FUNCTION "FC_WW_TELLER" : VOID
TITLE =
//$Revision: 1.56 $
//$Date: 2008/09/09 10:15:54CEST $
//$Author: schmoelp $
//
// Werkzeugwechsler Teller
AUTHOR : PS
FAMILY : DMC_H
NAME : WWPICKUP
VERSION : 0.0


VAR_INPUT
  gespannt : BOOL ;	// gespannt mit oder ohne Werkzeug
  gespannt_mWz : BOOL ;	// gespannt mit Werkzeug
  gespannt_oWz : BOOL ;	// gespannt ohne Werkzeug
  gespannt_Frg_Sp : BOOL ;	// gespannt mit Werkzeug Freigabe Spindeldrehen
  IB_MagKontr_aus : BOOL ;	//IB-Bit: Belegungskontrolle Magazin ausblenden
  AB_mit_Entriegeln : BOOL ;	//Ausbaustufe gesteuertes entriegeln im Magazin
  Frg_Service : BOOL ;	//Freigabe der Einzelbewegungen ohne Bedingung
  Bild_MAGEinstellung : BOOL ;
END_VAR
VAR_TEMP
  Klappe_auf_1 : BOOL ;
  Klappe_auf_2 : BOOL ;
  Vorbedingung_AF1 : BOOL ;
  Vorbedingung_AF2 : BOOL ;
  Vorbedingung_AF3 : BOOL ;
  PruefeAblageplatz : BOOL ;
  PruefeAbholplatz : BOOL ;
  ZvonPLC : BOOL ;
  IKZ_ausblasen : BOOL ;
  FC18_Error : BOOL ;
  Klappe_auf_BBK : BOOL ;
  Reset_Prgende : BOOL ;
  WV_laden_M1_aktiv : BOOL ;
  Schritt_gesetzt : BOOL ;
  Bild_WW_Handbedienung : BOOL ;
  MSST_Reset : BOOL ;
  WW_von_WZV : BOOL ;
  WZM_Fahrbefehl : BOOL ;
  BA_3_4 : BOOL ;
  F_ZHub_n_ausgefahren : BOOL ;
  F_ZHub_n_eingefahren : BOOL ;
  F_Mag_n_in_Position : BOOL ;
  F_Zange_n_auf : BOOL ;
  F_Zange_n_zu : BOOL ;
  F_Spanner_n_zu : BOOL ;
  F_Spanner_n_auf : BOOL ;
  F_Sp_n_gerichtet : BOOL ;
  F_MagKlappe_n_auf : BOOL ;
  F_MagKlappe_n_zu : BOOL ;
  F_Spindel_leer : BOOL ;
  F_VSP_Y_WW : BOOL ;
  HalterSp_auf : BOOL ;
  HalterSp_zu : BOOL ;
  PI_WZ_LS_GST : BOOL ;	//Positive Flanke Grundstellung Werkzeug entriegeln Ladestation
  FRG_WZ_MAN_RELEASE : BOOL ;
  Frg_Ventil_Hub : BOOL ;
  t_PI_T_quitt_Entladen : BOOL ;
  AB_WZB : BOOL ;	//mechanische Bruchkontrolle
  SFC12_RET_VAL : INT ;
  SFC12_SRCBLK : INT ;
  SFC12_DSTBLK : INT ;
  Achssperre : BOOL ;
  NewToolTx : BOOL ;
  NewToolT0 : BOOL ;
  OldToolTx : BOOL ;
  OldToolT0 : BOOL ;
  Schritt_vorwaerts : BOOL ;	//Schrittkette vorwärts
  Schritt_rueckwaerts : BOOL ;	//Schrittkette rückwärts
  Taste_vorwaerts : BOOL ;
  Taste_rueckwaerts : BOOL ;
  PI_T_vorwaerts : BOOL ;
  PI_T_rueckwaerts : BOOL ;
  EB_Frg_Klappe_auf : BOOL ;
  EB_Klappe_auf : BOOL ;
  EB_Frg_Klappe_zu : BOOL ;
  EB_Klappe_zu : BOOL ;
  EB_Frg_Wz_aus : BOOL ;
  EB_Frg_Wz_ein : BOOL ;
  EB_Frg_entspannen : BOOL ;
  EB_entspannen : BOOL ;
  EB_Frg_spannen : BOOL ;
  EB_spannen : BOOL ;
  EB_Frg_KR_einfahren : BOOL ;
  EB_KR_einfahren : BOOL ;
  EB_Frg_KR_ausfahren : BOOL ;
  EB_KR_ausfahren : BOOL ;
  EB_Frg_X_WWPos : BOOL ;
  EB_Frg_X_WartePos : BOOL ;
  EB_Hand_WW : BOOL ;
  Handbetrieb : BOOL ;
  Achse_angewaehlt : BOOL ;
  PI_Start_KR : BOOL ;
  Temp_INT : INT ;
  VSP_M_Wechsler : BOOL ;
  VSP_M_KR_GRSTn : BOOL ;
  VSP_M_Ls_GRSTn : BOOL ;
  VSP_M_BBK : BOOL ;
  VSP_M_aus_n : BOOL ;
  EB_Taste_steht_an : BOOL ;
  FC21_Error : BOOL ;
  t_AxFrg_y : BOOL ;
  t_Fahrbefehl_y : BOOL ;
  TX_O_WW_1_ZYL_GST : BOOL ;
  TX_O_WW_1_ZYL_SPI : BOOL ;
  A_DPR : ARRAY  [0 .. 15 ] OF BOOL ;
  FC21_ErrCode : INT ;
END_VAR
BEGIN
NETWORK
TITLE ============ allgemeine Signale ==============
// Netzwerk-Übersicht
// ==================
// NW 1: =========== allgemeine Signale ==============
// NW 2: Ausbaustufe mechanische Werkzeugbruchkontrolle
// NW 3: Taste Reset oder Programmende
// NW 4: Betriebsart 3, 4
// NW 5: JOG-Betrieb
// NW 6: Bildanwahl Einzelbewegung
// NW 7: Bildanwahl Semifunktion
// NW 8: Zange geöffnet
// NW 9: Zange geschlossen
// NW 10: Fahrbefehl Werkzeugmagazin steht an
// NW 11: ========== Signale von Werkzeugverwalung ==============
// NW 12: WZV: Werkzeugwechsel steht an
// NW 13: WZV: Aufgerufenes Werkzeug Tx
// NW 14: WZV: Aufgerufenes Werkzeug T0
// NW 15: WZV: Spindel belegt
// NW 16: WZV: Spindel leer
// NW 17: WZV: Vorbedingung Folge 1 Tx M6 Spindel leer
// NW 18: WZV: Vorbedingung Folge 2 Tx M6 Spindel belegt
// NW 19: WZV: Vorbedingung Folge 3 T0 M6 Spindel belegt
// NW 20: ============= Kegelreinigung ==================
// NW 21: KR: Einzelbewegung Freigabe einfahren
// NW 22: KR: Einzelbewegung einfahren
// NW 23: KR: Einzelbewegung Freigabe ausfahren
// NW 24: KR: Einzelbewegung ausfahren
// NW 25: KR: Einzelbewegung ausfahren speichern
// NW 26: KR: Einzelbewegung Ansteuerung Anzeige
// NW 27: Überwachung Kegelreinigung
// NW 28: KR: Start Werkzeug reinigen Tellermagazin
// NW 29: KR: aus-/einfahren
// NW 30: KR: Ausgang ausfahren
// NW 31: KR: Zeit starten
// NW 32: KR: beendet
// NW 33: ============== Werkzeugwechsel ===============
// NW 34: WW: Zyklus L6 wurde gestartet
// NW 35: WW: rücksetzen
// NW 36: WW: Auswertung Schritt gesetzt
// NW 37: WW: START
// NW 38: WW: Rücksetzen M-Funktion M06
// NW 39: WZW: Aktiver Ablauf
// NW 40: WW: 2nd software limit switch plus
// NW 41: WW: Folge 1 Tx M6 Spindel leer / Auftrag 1
// NW 42: WW: Folge 1 Freigabe fahre ins Magazin
// NW 43: WW: Folge 1 Auftrag 2: Einwechseln neues Werkzeug
// NW 44: WW: Folge 1 Tx M6 Spindel leer beendet
// NW 45: WW: Folge 2 Tx M6 Spindel belegt / Auftrag 3
// NW 46: WW: Folge 2 Freigabe fahre ins Magazin
// NW 47: WW: Folge 2 HILFSSCHRITT2
// NW 48: WW: Folge 2 Auftrag 2: Einwechseln neues Werkzeug
// NW 49: WW: Folge 2 beendet
// NW 50: WW: Folge 3 T0 M6 Spindel belegt / Auftrag 3
// NW 51: WW: Folge 3 Freigabe fahre ins Magazin
// NW 52: WW: Folge 3 Einwechseln kein Werkzeug
// NW 53: WW: Folge 3 beendet
// NW 54: WW: ABBRUCH -> FREIFAHREN
// NW 55: Taste Werkzeugwechsler vorwärts in Grundstellung fahren
// NW 56: Taste Werkzeugwechsler rückwärts in Grundstellung fahren
// NW 57: WW: Vorwärts Taste
// NW 58: WW: Rückwärts Taste
// NW 59: WW: Freigabe VOR/ZURUECK Freifahren
// NW 60: WW: Vorwärts Flanke Taste
// NW 61: WW: Vorwärts Bewegung
// NW 62: WW: Vorwärts Schrittkette
// NW 63: WW: Rückwärts Flanke Taste
// NW 64: WW: Rückwärts Bewegung
// NW 65: WW: Rückwärts gespeichert
// NW 66: WW: Rückwärts Schrittkette
// NW 67: WW: FREIGABE AUSGAENGE FUER ABLAUF
// NW 68: WW: ANZEIGE VORWAERTS
// NW 69: WW: ANZEIGE RUECKWAERTS
// NW 70: WW: Semifunktion Ansteuerung Anzeige Werkzeugwechsler
// NW 71: WW: initialisieren
// NW 72: WW: SCHRITT_0 GRUNDSTELLUNG
// NW 73: WW: GRUNDSTELLUNG MELDEN
// NW 74: WW: Grundstellung Werkzeugwechsler
// NW 75: WW: Werkzeugwechsel beendet an andere Module
// NW 76: WW: SCHRITT_1
// NW 77: WW: SCHRITT_2
// NW 78: WW: SCHRITT_3
// NW 79: WW: SCHRITT_4
// NW 80: WW: Datentausch ablegen
// NW 81: WW: SCHRITT_5
// NW 82: WW: SCHRITT_6
// NW 83: WW: SCHRITT_7 SONDERSCHRITT
// NW 84: WW: Rücksetzen Auftrag 1 und 3
// NW 85: WW: SCHRITT_8
// NW 86: WW: SCHRITT_9
// NW 87: WW: Datentausch aufnehmen
// NW 88: WW: SCHRITT_10
// NW 89: WW: SCHRITT_11
// NW 90: WW: Rücksetzen Schritt 10
// NW 91: WW: SCHRITT_12
// NW 92: WW: Prüfen, ob Ablageplatz im Magazin leer ist
// NW 93: WW: Prüfen, ob Abholplatz im Magazin belegt ist
// NW 94: WW: Magazinplatz Belegung kontrolliert und i.O.
// NW 95: =========== Magazinklappe (Werkzeugwechslertür) =============
// NW 96: WWT: öffnen mit Freigabe
// NW 97: WWT: öffnen ohne Freigabe
// NW 98: WWT: Einzelbewegung Freigabe öffnen
// NW 99: WWT: Einzelbewegung öffnen
// NW 100: WWT: Einzelbewegung Freigabe schliessen
// NW 101: WWT: Einzelbewegung schliessen
// NW 102: WWT: Einzelbewegung öffnen speichern
// NW 103: WWT: Einzelbewegung schliessen speichern
// NW 104: WWT: Einzelbewegung Ansteuerung Anzeige
// NW 105: HMI-Bild 35 (WZW7): WWT: Einzelbewegung Ansteuerung Anzeige
// NW 106: WWT: Ausgang öffnen
// NW 107: WWT: Ausgang schliessen
// NW 108: WWT: Ausgang schliessen Reset M272
// NW 109: WWT: Reset Ausgang schliessen
// NW 110: ========== Werkzeug in / aus Spindel ===============
// NW 111: WZHUB: BEFEHL FAHRE auf AUSFAHRPOSITION
// NW 112: WZHUB: BEFEHL FAHRE WW-Achse auf Einfahrposition
// NW 113: Hub in Spindelstellung
// NW 114: Hub in Grundstellung
// NW 115: WZHUB: Einzelbewegung Freigabe Werkzeug Spindel aus- einfahren
// NW 116: WZHUB: Einzelbewegung Werkzeug aus Spindel ausfahren
// NW 117: WZHUB: Einzelbewegung WW-Achse auf Einfahrposition
// NW 118: WZHUB: Reset Einzelbewegung WW-Achse wenn nicht in Position
// NW 119: WZHUB: Freigabe Ansteuerung Ventil Hub ein- / ausfahren
// NW 120: WZHUB: Ventil Hub einfahren
// NW 121: WZHUB: Ventil Hub ausfahren
// NW 122: WZHUB: (WZW1) Einzelbewegung Ansteuerung Anzeige
// NW 123: WZHUB: (WZW7) Einzelbewegung Ansteuerung Anzeige
// NW 124: =========== Spindel in / aus Werkzeugwechsler ============
// NW 125: X-Achse: Befehl auf Warteposition fahren
// NW 126: X-Achse: Befehl auf Wechselposition fahren
// NW 127: X-Achse: Einzelbewegung Freigabe auf Warteposition
// NW 128: X-Achse: Einzelbewegung auf Warteposition fahren
// NW 129: X-Achse: Einzelbewegung Freigabe auf Wechselposition
// NW 130: X-Achse: Einzelbewegung auf Wechselposition fahren
// NW 131: X-Achse: Einzelbewegung Ansteuerung Anzeige
// NW 132: Y-Achse: Freigabe
// NW 133: Y-Achse: Fahrbefehl
// NW 134: Y-Achse: HMI Rettung
// NW 135: Spindel: Befehl auf Werkzeugwechselposition
// NW 136: Spindel: HMI Rettung
// NW 137: ======== Werkzeug im Magazin entsichern Wechselstelle ========
// NW 138: WW_MagTasche: BEFEHL Werkzeug entsichern Spindelseite
// NW 139: WW_MagTasche: Ausgang Werkzeug entsichern Spindelseite
// NW 140: ======== Werkzeug im Magazin entsichern Ladestelle ========
// NW 141: WM_MagTasche: Ausgang Werkzeug entsichern an BELADESTATION
// NW 142: WM_MagTasche: Werkzeug wurde an BELADESTATION entsichert
// NW 143: ========= Werkzeug entspannen im Ablauf ===========
// NW 144: WZ-Spanner: Einzelbewegung Freigabe Werkzeug entspannen
// NW 145: WZ-Spanner: Einzelbewegung Werkzeug entspannen
// NW 146: WZ-Spanner: Einzelbewegung Freigabe Werkzeug spannen
// NW 147: WZ-Spanner: Einzelbewegung Werkzeug spannen
// NW 148: WZ-Spanner: Einzelbewegung Ansteuerung Anzeige
// NW 149: WZ-Spanner: Einzelbewegung Ansteuerung Anzeige
// NW 150: WZ-Spanner: BEFEHL WZ ENTSPANNEN
// NW 151: WZ-Spanner: BEFEHL WZ SPANNEN
// NW 152: WZ-Spanner: Ausgang Spanner öffnen
// NW 153: Ausgang SPINDELKONUS AUSBLASEN
// NW 154: Positive Flanke Taste quittieren Entladen
// NW 155: Pneumatikzyl. Verriegelung WZ lösen
// NW 156: Pneumatikzyl. Verriegelung WZ verriegeln
// NW 157: ========= Vorschubsperren ===============
// NW 158: VSP, alle Achsen
// NW 159: VSP-X, Werkzeugwechsler
// NW 160: _701303 Vorschubsperre X Werkzeugwechsler
// NW 161: VSP-Y, Werkzeugwechsler
// NW 162: Fehler Vorschubsperre Y Werkzeugwechsler
// NW 163: VSP-Z, Werkzeugwechsler
// NW 164: _701305 Vorschubsperre Z Werkzeugwechsler
// NW 165: VSP-M, Bohrerbruchkontrolle nicht in Grundstellung
// NW 166: VSP-M, Magazin nicht in Position aus Spindel ausgefahren
// NW 167: VSP-M, Werkzeugwechsler
// NW 168: VSP-M, Waschstation nicht in Grundstellung
// NW 169: Positive Flanke Grundstellung Werkzeug entriegeln Ladestation
// NW 170: Werkzeug wurde richtig eingelegt
// NW 171: VSP-M, Werkzeug in Ladestation nicht gesichert
// NW 172: VSP-M, Werkzeugwechsler
// NW 173: VSP-M, Verzögerung Fehlermeldung
// NW 174: 701306 "MEL, Vorschubsperre Magazin Werkzeugwechsler"
// NW 175: 701307 Vorschubsperre Magazin Waschstation nicht in Grundst
// NW 176: 701308 VSP Magazin Bohrerbruchkontrolle nicht in Grundstellung
// NW 177: 701309 VSP, Magazin nicht in Position aus Spindel ausgefahren
// NW 178: 700363 Warnung: Werkzeug in Ladestation nicht gesichert
// NW 179: 511214: Meldung: Werkzeug in Ladestation nicht gesichert
// NW 180: _700434 VS-H, ENDSCHALTERSTOERUNG Werkzeugwechsel
// NW 181: ============ Überwachung Endposition ==========
// NW 182: Fehler MAGAZIN NICHT AUSGEFAHREN
// NW 183: Fehler MAGAZIN NICHT EINGEFAHREN
// NW 184: Fehler MAGAZIN NICHT IN POSITION
// NW 185: Fehler WZ-ZANGE NICHT OFFEN
// NW 186: Fehler WZ-ZANGE NICHT GESCHLOSSEN
// NW 187: Fehler WZ-SPANNER NICHT GESPANNT
// NW 188: Fehler WZ-SPANNER NICHT GELOEST
// NW 189: Fehler SPINDEL NICHT GERICHTET
// NW 190: Fehler Magazinklappe nicht geöffnet
// NW 191: Fehler Magazinklappe nicht geschlossen
// NW 192: Fehler Spindel leer
// NW 193: gespeicherte Fehlermeldungen löschen
// NW 194: WZW nicht erlaubt
// NW 195: Start Wartezeit für Endlagenkontrolle
// NW 196: Wartezeit für Endlagenkontrolle abgelaufen ?
// NW 197: _700355 Werkzeugmagazin nicht ausgefahren
// NW 198: _700356 Werkzeugmagazin nicht eingefahren
// NW 199: _700361 Magazin nicht in Position
// NW 200: _700354 Werkzeug im Magazin nicht entsichert
// NW 201: _700362 Werkzeug in Magazin nicht gesichert
// NW 202: _700353 Werkzeug in Spindel nicht gespannt
// NW 203: _700351 Werkzeug in Spindel nicht entspannt
// NW 204: _700360 Spindel nicht gerichtet
// NW 205: _700357 Magazinklappe nicht geöffnet
// NW 206: _700358 Magazinklappe nicht geschlossen
// NW 207: _701302 Spindel leer
// NW 208: _701304 VSP-Y Werkzeugwechsler
// NW 209: ======== Sonstige Fehler- Betriebsmeldungen ===========
// NW 210: _700348 Magazinplatz/Greifer belegt
// NW 211: _700349 Magazinplatz/Greifer leer
// NW 212: _700350 Ladestation nicht geschlossen
// NW 213: _701321 Spindel belegt
// NW 214: _700352 Werkzeug Be- oder Entladen aktiv
// NW 215: Taste für Einzelbewegung Achsen betätigt
// NW 216: _700550 EINLESESPERRE, Werkzeugwechsel
// NW 217: ======== ASUP Einzelbewegung Achsen ========
// NW 218: ASUP-EB: Schnittstelle Dual-Port-RAM 16.0
// NW 219: ASUP-EB: Schnittstelle Dual-Port-RAM 16.1
// NW 220: ASUP-EB: Schnittstelle Dual-Port-RAM 16.2
// NW 221: ASUP-EB: Schnittstelle Dual-Port-RAM 16.3
// NW 222: ASUP-EB: Schnittstelle Dual-Port-RAM 16.4
// NW 223: Asup abbrechen wenn Taste wieder losgelassen wird
// NW 224: Eingang "MSSTstReset" auf "1" zuweisen
// NW 225: ASUP-Rettung: Werkzeugwechsler automatisch in Grundstellung
// NW 226: ASUP-EB: Schnittstelle Dual-Port-RAM nicht benutzte Bits
// NW 227: ASUP-EB: Aufruf Kanal-DB für FC21
// NW 228: ASUP-EB: Übergabe an DUAL-PORT-RAM
// NW 229: ASUP-EB: Start für Einzelbewegung Achsen
// NW 230: GRundstelltung Radmagazin
// NW 231: ============ Signale an andere Module =============
// NW 232: Übergabe der Schrittnummer Werkzeugwechsel an HMI
// NW 233: An NC: PLC-Freigabe Werkzeugwechsel
// NW 234: An NC: Rad in Wechselstellung nach Be./Enladen an Beladestelle
//
      NOP   0;

NETWORK
TITLE =Ausbaustufe mechanische Werkzeugbruchkontrolle
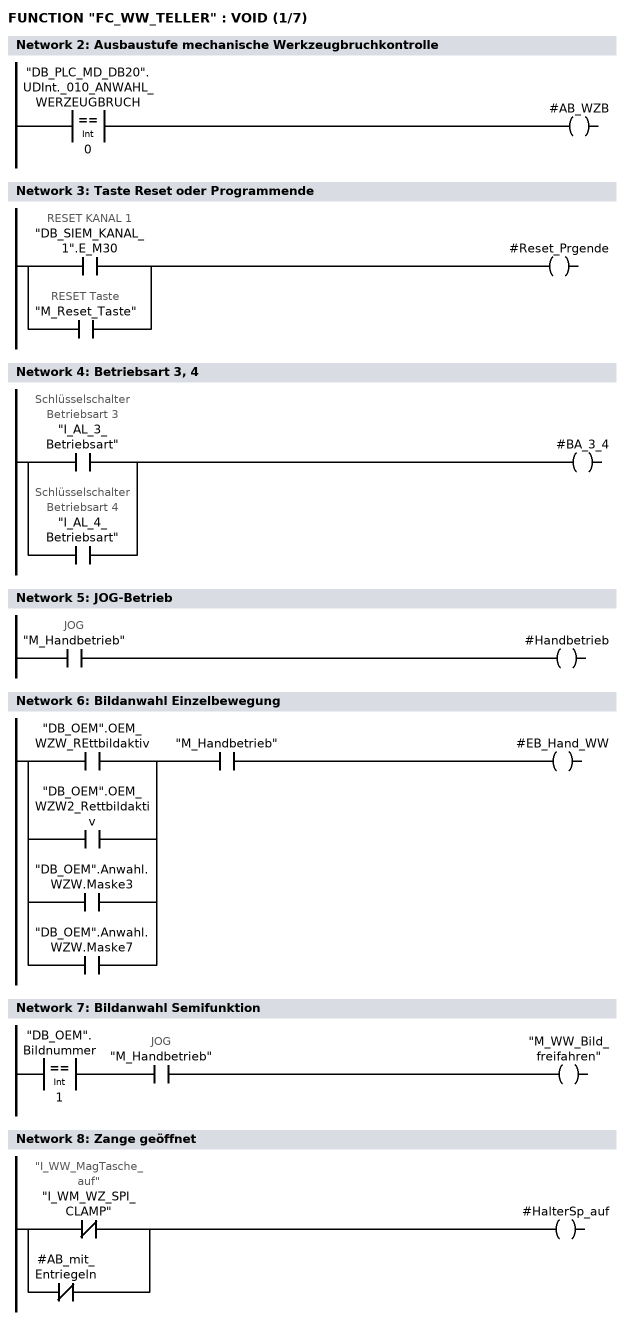

      L     "DB_PLC_MD_DB20".UDInt._010_ANWAHL_WERZEUGBRUCH;
      L     0;
      ==I   ;
      =     #AB_WZB;
NETWORK
TITLE =Taste Reset oder Programmende

      O     "DB_SIEM_KANAL_1".E_M30; // RESET KANAL 1
      O     "M_Reset_Taste"; // RESET Taste
      =     #Reset_Prgende;

NETWORK
TITLE =Betriebsart 3, 4

      O     "I_AL_3_Betriebsart"; // Schlüsselschalter Betriebsart 3
      O     "I_AL_4_Betriebsart"; // Schlüsselschalter Betriebsart 4
      =     #BA_3_4;


NETWORK
TITLE =JOG-Betrieb

      U     "M_Handbetrieb"; // JOG
      =     #Handbetrieb;

NETWORK
TITLE =Bildanwahl Einzelbewegung
//
      U(    ;
      O     "DB_OEM".OEM_WZW_REttbildaktiv;
      O     "DB_OEM".OEM_WZW2_Rettbildaktiv;
      O     "DB_OEM".Anwahl.WZW.Maske3;
      O     "DB_OEM".Anwahl.WZW.Maske7;
      )     ; // JOG
      U     "M_Handbetrieb";

      =     #EB_Hand_WW;
NETWORK
TITLE =Bildanwahl Semifunktion

      U(    ;
      L     "DB_OEM".Bildnummer;
      L     1;
      ==I   ;
      )     ;
      U     "M_Handbetrieb"; // JOG
      =     "M_WW_Bild_freifahren";

NETWORK
TITLE =Zange geöffnet

      ON    "I_WM_WZ_SPI_CLAMP"; //"I_WW_MagTasche_auf"
      ON    #AB_mit_Entriegeln;
      =     #HalterSp_auf;

NETWORK
TITLE =Zange geschlossen
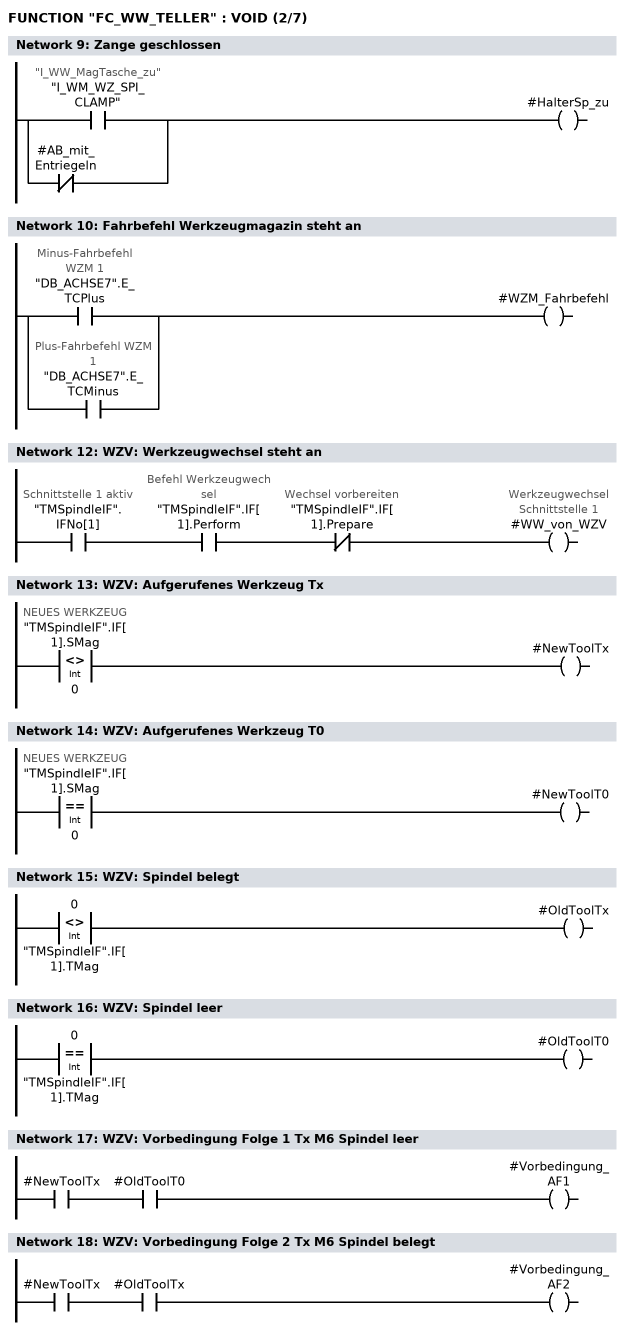

      O     "I_WM_WZ_SPI_CLAMP"; //"I_WW_MagTasche_zu"
      ON    #AB_mit_Entriegeln;
      =     #HalterSp_zu;

NETWORK
TITLE =Fahrbefehl Werkzeugmagazin steht an

      O     "DB_ACHSE7".E_TCPlus; // Minus-Fahrbefehl WZM 1
      O     "DB_ACHSE7".E_TCMinus; // Plus-Fahrbefehl WZM 1
      =     #WZM_Fahrbefehl;

NETWORK
TITLE =========== Signale von Werkzeugverwalung ==============



NETWORK
TITLE =WZV: Werkzeugwechsel steht an

      U     "TMSpindleIF".IFNo[1]; // Schnittstelle 1 aktiv
      U     "TMSpindleIF".IF[1].Perform; // Befehl Werkzeugwechsel
      UN    "TMSpindleIF".IF[1].Prepare; // Wechsel vorbereiten
      =     #WW_von_WZV; // Werkzeugwechsel Schnittstelle 1

NETWORK
TITLE =WZV: Aufgerufenes Werkzeug Tx

      L     "TMSpindleIF".IF[1].SMag; // NEUES WERKZEUG
      L     0;
      <>I   ;
      =     #NewToolTx;

NETWORK
TITLE =WZV: Aufgerufenes Werkzeug T0

      L     "TMSpindleIF".IF[1].SMag; // NEUES WERKZEUG
      L     0;
      ==I   ;
      =     #NewToolT0;

NETWORK
TITLE =WZV: Spindel belegt

      L     0;
      L     "TMSpindleIF".IF[1].TMag; // ALTES WERKZEUG
      <>I   ;
      =     #OldToolTx;

NETWORK
TITLE =WZV: Spindel leer

      L     0;
      L     "TMSpindleIF".IF[1].TMag; // ALTES WERKZEUG
      ==I   ;
      =     #OldToolT0;

NETWORK
TITLE =WZV: Vorbedingung Folge 1 Tx M6 Spindel leer

      U     #NewToolTx;
      U     #OldToolT0;
      =     #Vorbedingung_AF1;

NETWORK
TITLE =WZV: Vorbedingung Folge 2 Tx M6 Spindel belegt

      U     #NewToolTx;
      U     #OldToolTx;
      =     #Vorbedingung_AF2;
NETWORK
TITLE =WZV: Vorbedingung Folge 3 T0 M6 Spindel belegt
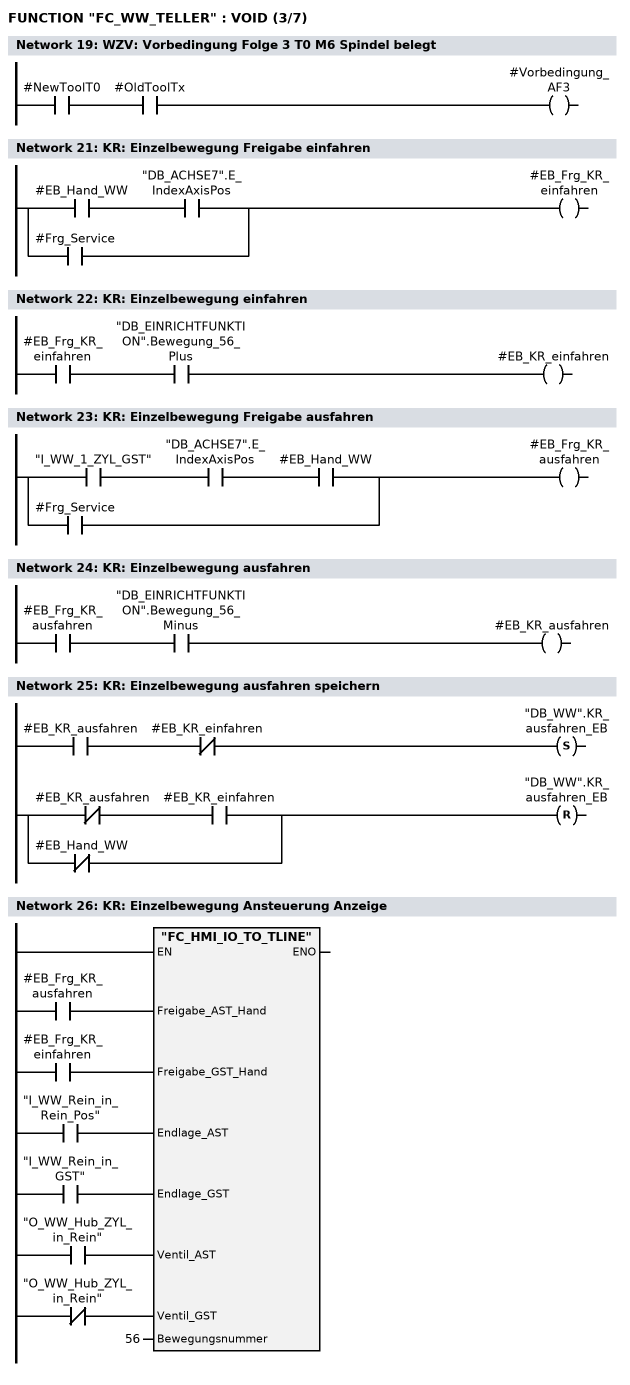

      U     #NewToolT0;
      U     #OldToolTx;
      =     #Vorbedingung_AF3;
NETWORK
TITLE ============== Kegelreinigung ==================



NETWORK
TITLE =KR: Einzelbewegung Freigabe einfahren

      U     #EB_Hand_WW;
      U     "DB_ACHSE7".E_IndexAxisPos;
      O     #Frg_Service;
      =     #EB_Frg_KR_einfahren;

NETWORK
TITLE =KR: Einzelbewegung einfahren

      U     #EB_Frg_KR_einfahren;
      U     "DB_EINRICHTFUNKTION".Bewegung_56_Plus;
      =     #EB_KR_einfahren;

NETWORK
TITLE =KR: Einzelbewegung Freigabe ausfahren

      U     "I_WW_1_ZYL_GST";
      U     "DB_ACHSE7".E_IndexAxisPos;
      U     #EB_Hand_WW;
      O     #Frg_Service;
      =     #EB_Frg_KR_ausfahren;
NETWORK
TITLE =KR: Einzelbewegung ausfahren

      U     #EB_Frg_KR_ausfahren;
      U     "DB_EINRICHTFUNKTION".Bewegung_56_Minus;
      =     #EB_KR_ausfahren;

NETWORK
TITLE =KR: Einzelbewegung ausfahren speichern

      U     #EB_KR_ausfahren;
      UN    #EB_KR_einfahren;
      S     "DB_WW".KR_ausfahren_EB;

      U(    ;
      UN    #EB_KR_ausfahren;
      U     #EB_KR_einfahren;
      ON    #EB_Hand_WW;
      )     ;
      R     "DB_WW".KR_ausfahren_EB;
      NOP   0;

NETWORK
TITLE =KR: Einzelbewegung Ansteuerung Anzeige

      U     #EB_Frg_KR_ausfahren;
      =     L     24.0;
      BLD   103;
      U     #EB_Frg_KR_einfahren;
      =     L     24.1;
      BLD   103;
      U     "I_WW_Rein_in_Rein_Pos";
      =     L     24.2;
      BLD   103;
      U     "I_WW_Rein_in_GST";
      =     L     24.3;
      BLD   103;
      U     "O_WW_Hub_ZYL_in_Rein";
      =     L     24.4;
      BLD   103;
      UN    "O_WW_Hub_ZYL_in_Rein";
      =     L     24.5;
      BLD   103;
      CALL "FC_HMI_IO_TO_TLINE" (
           Freigabe_AST_Hand        := L     24.0,
           Freigabe_GST_Hand        := L     24.1,
           Endlage_AST              := L     24.2,
           Endlage_GST              := L     24.3,
           Ventil_AST               := L     24.4,
           Ventil_GST               := L     24.5,
           Bewegungsnummer          := 56);
      NOP   0;
NETWORK
TITLE =Überwachung Kegelreinigung
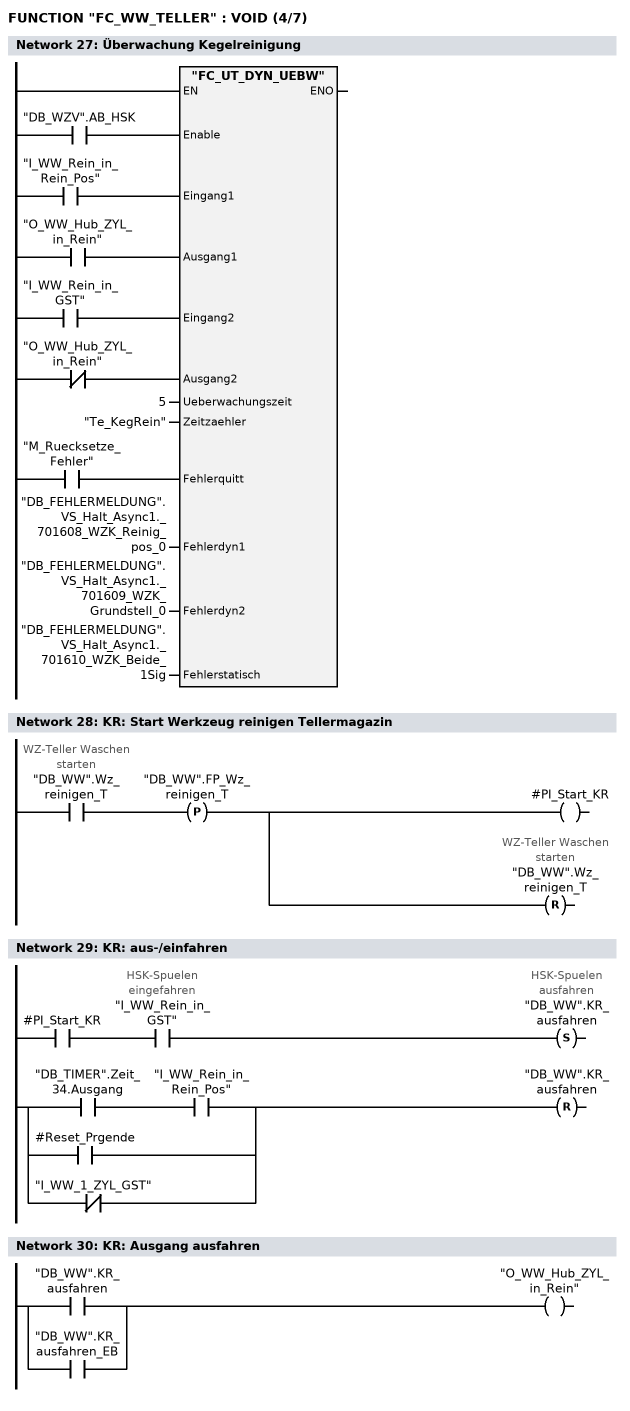

      U     "DB_WZV".AB_HSK;
      =     L     24.0;
      BLD   103;
      U     "I_WW_Rein_in_Rein_Pos";
      =     L     24.1;
      BLD   103;
      U     "O_WW_Hub_ZYL_in_Rein";
      =     L     24.2;
      BLD   103;
      U     "I_WW_Rein_in_GST";
      =     L     24.3;
      BLD   103;
      UN    "O_WW_Hub_ZYL_in_Rein";
      =     L     24.4;
      BLD   103;
      U     "M_Ruecksetze_Fehler";
      =     L     24.5;
      BLD   103;
      CALL "FC_UT_DYN_UEBW" (
           Enable                   := L     24.0,
           Eingang1                 := L     24.1,
           Ausgang1                 := L     24.2,
           Eingang2                 := L     24.3,
           Ausgang2                 := L     24.4,
           Ueberwachungszeit        := 5,
           Zeitzaehler              := "Te_KegRein",
           Fehlerquitt              := L     24.5,
           Fehlerdyn1               := "DB_FEHLERMELDUNG".VS_Halt_Async1._701608_WZK_Reinig_pos_0,
           Fehlerdyn2               := "DB_FEHLERMELDUNG".VS_Halt_Async1._701609_WZK_Grundstell_0,
           Fehlerstatisch           := "DB_FEHLERMELDUNG".VS_Halt_Async1._701610_WZK_Beide_1Sig);
      NOP   0;
NETWORK
TITLE =KR: Start Werkzeug reinigen Tellermagazin

      U     "DB_WW".Wz_reinigen_T; // WZ-Teller Waschen starten
      FP    "DB_WW".FP_Wz_reinigen_T; // PF: WZ waschen Start
      =     #PI_Start_KR;
      R     "DB_WW".Wz_reinigen_T; // WZ-Teller Waschen starten

NETWORK
TITLE =KR: aus-/einfahren

      U     #PI_Start_KR;
      U     "I_WW_Rein_in_GST"; // HSK-Spuelen eingefahren
      S     "DB_WW".KR_ausfahren; // HSK-Spuelen ausfahren

      U(    ;
      U     "DB_TIMER".Zeit_34.Ausgang;
      U     "I_WW_Rein_in_Rein_Pos";
      O     #Reset_Prgende;

      ON    "I_WW_1_ZYL_GST";
      )     ;
      R     "DB_WW".KR_ausfahren;
      NOP   0;
NETWORK
TITLE =KR: Ausgang ausfahren

      O     "DB_WW".KR_ausfahren;
      O     "DB_WW".KR_ausfahren_EB;
      =     "O_WW_Hub_ZYL_in_Rein";

NETWORK
TITLE =KR: Zeit starten
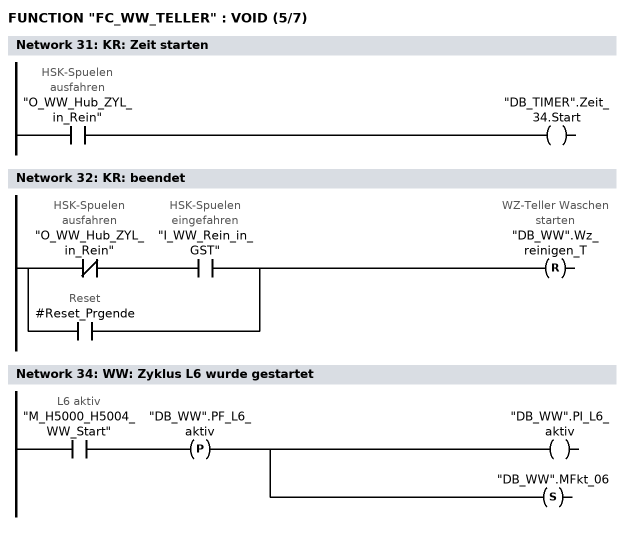

      U     "O_WW_Hub_ZYL_in_Rein"; // HSK-Spuelen ausfahren
      =     "DB_TIMER".Zeit_34.Start;

NETWORK
TITLE =KR: beendet

      UN    "O_WW_Hub_ZYL_in_Rein"; // HSK-Spuelen ausfahren
      U     "I_WW_Rein_in_GST"; // HSK-Spuelen eingefahren
      O     #Reset_Prgende; //Reset
      R     "DB_WW".Wz_reinigen_T; // WZ-Teller Waschen starten

NETWORK
TITLE =============== Werkzeugwechsel ===============



NETWORK
TITLE =WW: Zyklus L6 wurde gestartet

      U     "M_H5000_H5004_WW_Start"; // L6 aktiv
      FP    "DB_WW".PF_L6_aktiv;
      =     "DB_WW".PI_L6_aktiv;
      S     "DB_WW".MFkt_06;

NETWORK
TITLE =WW: rücksetzen
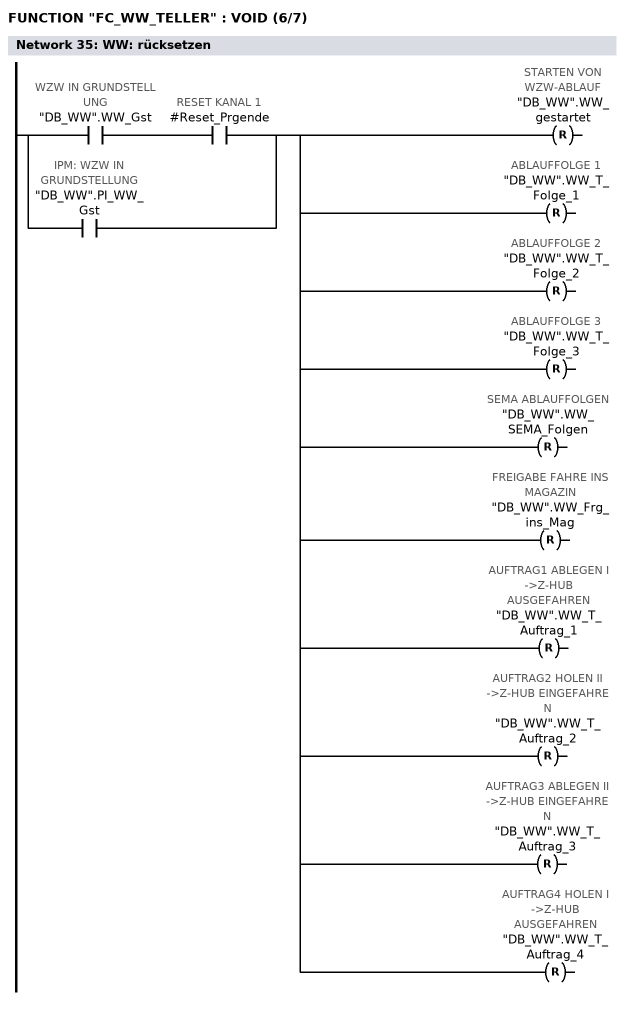

      U     "DB_WW".WW_Gst; // WZW IN GRUNDSTELLUNG
      U     #Reset_Prgende; // RESET KANAL 1
      O     "DB_WW".PI_WW_Gst; // IPM: WZW IN GRUNDSTELLUNG
      R     "DB_WW".WW_gestartet; // STARTEN VON WZW-ABLAUF
      R     "DB_WW".WW_T_Folge_1; // ABLAUFFOLGE 1
      R     "DB_WW".WW_T_Folge_2; // ABLAUFFOLGE 2
      R     "DB_WW".WW_T_Folge_3; // ABLAUFFOLGE 3
      R     "DB_WW".WW_SEMA_Folgen; // SEMA ABLAUFFOLGEN
      R     "DB_WW".WW_Frg_ins_Mag; // FREIGABE FAHRE INS MAGAZIN
      R     "DB_WW".WW_T_Auftrag_1; // AUFTRAG1 ABLEGEN I ->Z-HUB AUSGEFAHREN
      R     "DB_WW".WW_T_Auftrag_2; // AUFTRAG2 HOLEN II ->Z-HUB EINGEFAHREN
      R     "DB_WW".WW_T_Auftrag_3; // AUFTRAG3 ABLEGEN II ->Z-HUB EINGEFAHREN
      R     "DB_WW".WW_T_Auftrag_4; // AUFTRAG4 HOLEN I ->Z-HUB AUSGEFAHREN

NETWORK
TITLE =WW: Auswertung Schritt gesetzt
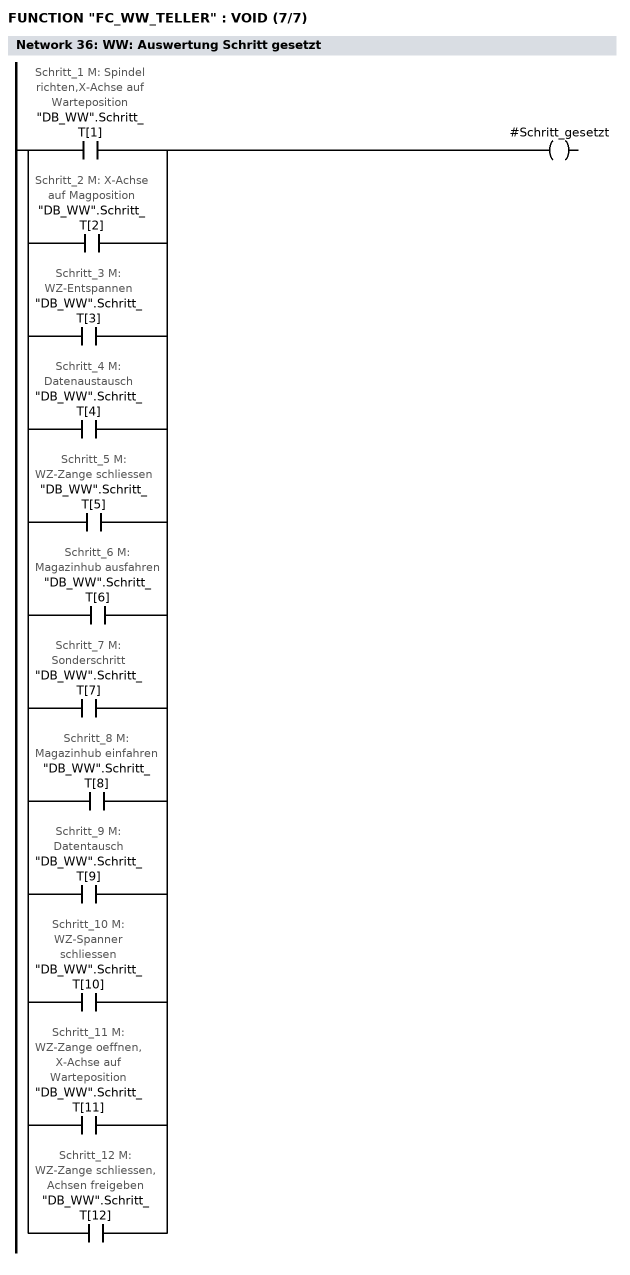

      O     "DB_WW".Schritt_T[1]; // Schritt_1 M: Spindel richten,X-Achse auf Warteposition
      O     "DB_WW".Schritt_T[2]; // Schritt_2 M: X-Achse auf Magposition
      O     "DB_WW".Schritt_T[3]; // Schritt_3 M: WZ-Entspannen
      O     "DB_WW".Schritt_T[4]; // Schritt_4 M: Datenaustausch
      O     "DB_WW".Schritt_T[5]; // Schritt_5 M: WZ-Zange schliessen
      O     "DB_WW".Schritt_T[6]; // Schritt_6 M: Magazinhub ausfahren
      O     "DB_WW".Schritt_T[7]; // Schritt_7 M: Sonderschritt
      O     "DB_WW".Schritt_T[8]; // Schritt_8 M: Magazinhub einfahren
      O     "DB_WW".Schritt_T[9]; // Schritt_9 M: Datentausch
      O     "DB_WW".Schritt_T[10]; // Schritt_10 M: WZ-Spanner schliessen
      O     "DB_WW".Schritt_T[11]; // Schritt_11 M: WZ-Zange oeffnen, X-Achse auf Warteposition
      O     "DB_WW".Schritt_T[12]; // Schritt_12 M: WZ-Zange schliessen, Achsen freigeben
      =     #Schritt_gesetzt;

NETWORK
TITLE =WW: START

      UN(   ;
      U(    ;
      L     "TMSpindleIF".IF[1].SMag; // NEUES WERKZEUG
      L     9999;
      ==I   ;
      )     ;
      U(    ;
      L     "TMSpindleIF".IF[1].TMag; // ALTES WERKZEUG
      L     0;
      ==I   ;
      )     ;
      O     ;
      U(    ;
      L     "TMSpindleIF".IF[1].SMag; // NEUES WERKZEUG
      L     9999;
      ==I   ;
      )     ;
      U(    ;
      L     "TMSpindleIF".IF[1].TMag; // ALTES WERKZEUG
      L     9999;
      ==I   ;
      )     ;
      )     ;
      U     "DB_WW".MFkt_06;
      UN    "DB_WW".PI_WW_Gst;
      U     "DB_WW".WW_Gst;
      UN    "DB_WZV".Mag1_Laden_aktiv;
      U     "DB_WZV".Mag1_inPos_WST;
      U     "I_WM_Energiefreigabe";
      UN    "DB_WW".WW_gestartet;
      O     #Schritt_gesetzt;
      S     "DB_WW".WW_gestartet;
NETWORK
TITLE =WW: Rücksetzen M-Funktion M06
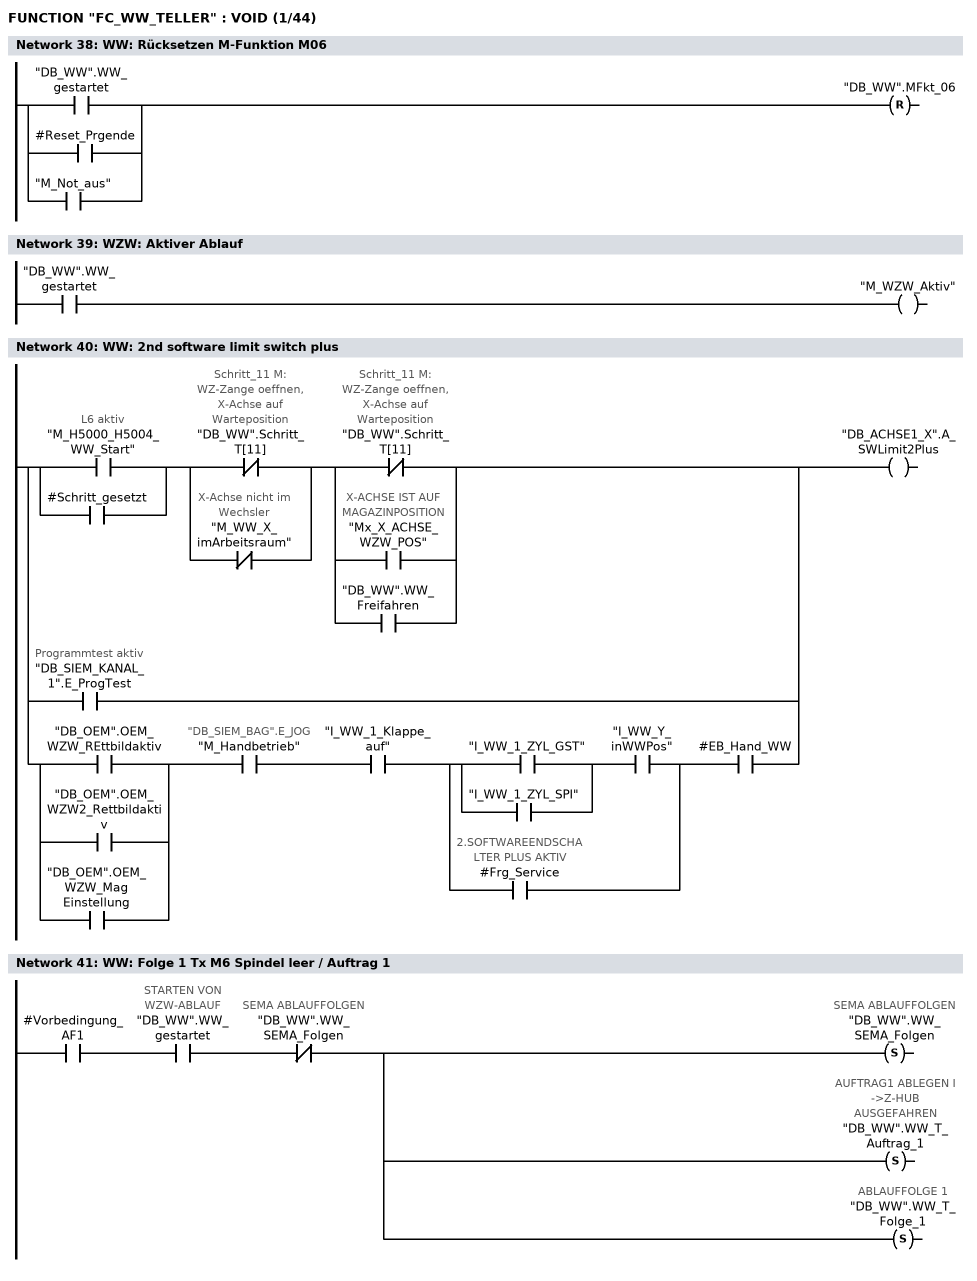

      O     "DB_WW".WW_gestartet;
      O     #Reset_Prgende;
      O     "M_Not_aus";
      R     "DB_WW".MFkt_06;
NETWORK
TITLE =WZW: Aktiver Ablauf

      U     "DB_WW".WW_gestartet;
      =     "M_WZW_Aktiv";

NETWORK
TITLE =WW: 2nd software limit switch plus

      U(    ;
      O     "M_H5000_H5004_WW_Start"; // L6 aktiv
      O     #Schritt_gesetzt;
      )     ;
      U(    ;
      ON    "DB_WW".Schritt_T[11]; // Schritt_11 M: WZ-Zange oeffnen, X-Achse auf Warteposition
      ON    "M_WW_X_imArbeitsraum"; // X-Achse nicht im Wechsler
      )     ;
      U(    ;
      ON    "DB_WW".Schritt_T[11]; // Schritt_11 M: WZ-Zange oeffnen, X-Achse auf Warteposition
      O     "Mx_X_ACHSE_WZW_POS"; // X-ACHSE IST AUF MAGAZINPOSITION
      O     "DB_WW".WW_Freifahren;
      )     ;

      O     "DB_SIEM_KANAL_1".E_ProgTest; // Programmtest aktiv
      O     ;
      U(    ;
      O     "DB_OEM".OEM_WZW_REttbildaktiv;
      O     "DB_OEM".OEM_WZW2_Rettbildaktiv;
      O     "DB_OEM".OEM_WZW_MagEinstellung;
      )     ;
      U     "M_Handbetrieb"; // "DB_SIEM_BAG".E_JOG
//    U     "DB_EINRICHTFUNKTION".Bewegung_14_Plus
      U     "I_WW_1_Klappe_auf";
      U(    ;
      U(    ;
      O     "I_WW_1_ZYL_GST";
      O     "I_WW_1_ZYL_SPI";
      )     ;
      U     "I_WW_Y_inWWPos";
      O     #Frg_Service; // 2.SOFTWAREENDSCHALTER PLUS AKTIV

      )     ;
      U     #EB_Hand_WW;
      =     "DB_ACHSE1_X".A_SWLimit2Plus;
NETWORK
TITLE =WW: Folge 1 Tx M6 Spindel leer / Auftrag 1

      U     #Vorbedingung_AF1;
      U     "DB_WW".WW_gestartet; // STARTEN VON WZW-ABLAUF
      UN    "DB_WW".WW_SEMA_Folgen; // SEMA ABLAUFFOLGEN
      S     "DB_WW".WW_SEMA_Folgen; // SEMA ABLAUFFOLGEN
      S     "DB_WW".WW_T_Auftrag_1; // AUFTRAG1 ABLEGEN I ->Z-HUB AUSGEFAHREN
      S     "DB_WW".WW_T_Folge_1; // ABLAUFFOLGE 1

NETWORK
TITLE =WW: Folge 1 Freigabe fahre ins Magazin
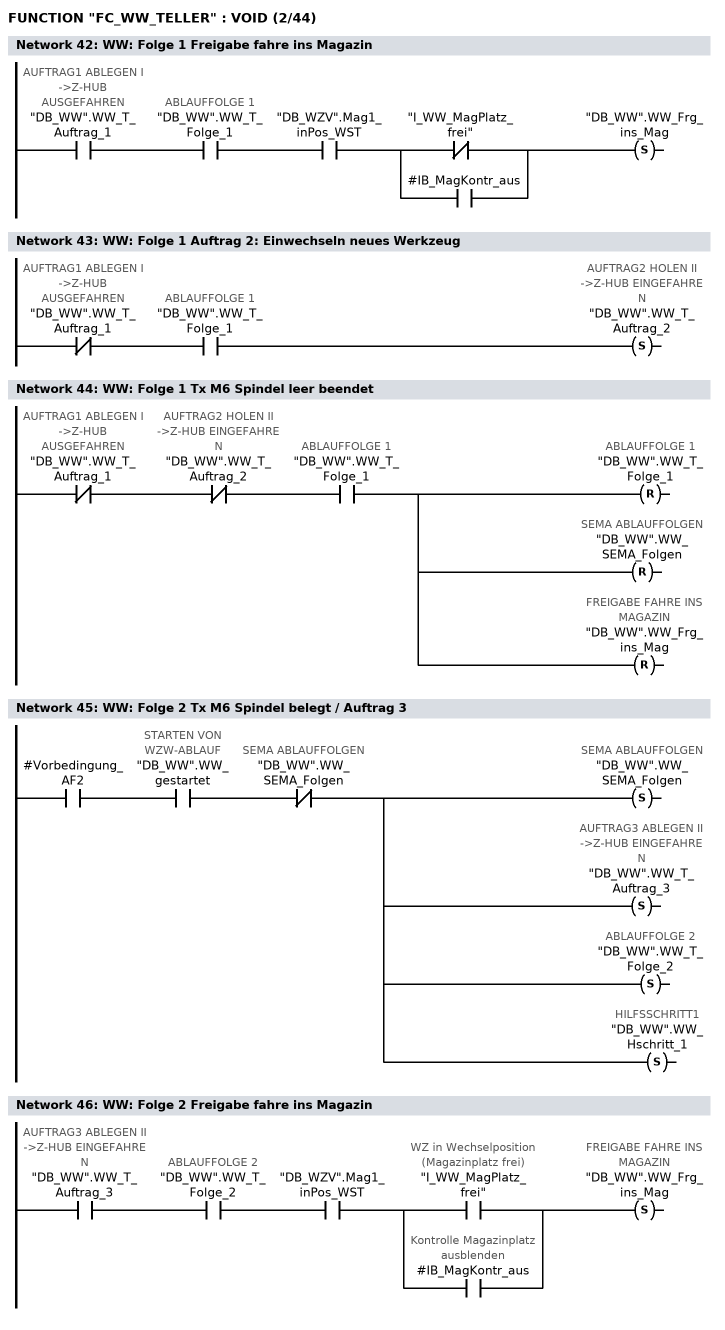

      U     "DB_WW".WW_T_Auftrag_1; // AUFTRAG1 ABLEGEN I ->Z-HUB AUSGEFAHREN
      U     "DB_WW".WW_T_Folge_1; // ABLAUFFOLGE 1
      U     "DB_WZV".Mag1_inPos_WST;
      U(    ; // FREIGABE FAHRE INS MAGAZIN

      ON    "I_WW_MagPlatz_frei";
      O     #IB_MagKontr_aus;
      )     ;
      S     "DB_WW".WW_Frg_ins_Mag;
NETWORK
TITLE =WW: Folge 1 Auftrag 2: Einwechseln neues Werkzeug

      UN    "DB_WW".WW_T_Auftrag_1; // AUFTRAG1 ABLEGEN I ->Z-HUB AUSGEFAHREN
      U     "DB_WW".WW_T_Folge_1; // ABLAUFFOLGE 1
      S     "DB_WW".WW_T_Auftrag_2; // AUFTRAG2 HOLEN II ->Z-HUB EINGEFAHREN

NETWORK
TITLE =WW: Folge 1 Tx M6 Spindel leer beendet

      UN    "DB_WW".WW_T_Auftrag_1; // AUFTRAG1 ABLEGEN I ->Z-HUB AUSGEFAHREN
      UN    "DB_WW".WW_T_Auftrag_2; // AUFTRAG2 HOLEN II ->Z-HUB EINGEFAHREN
      U     "DB_WW".WW_T_Folge_1; // ABLAUFFOLGE 1
      R     "DB_WW".WW_T_Folge_1; // ABLAUFFOLGE 1
      R     "DB_WW".WW_SEMA_Folgen; // SEMA ABLAUFFOLGEN
      R     "DB_WW".WW_Frg_ins_Mag; // FREIGABE FAHRE INS MAGAZIN

NETWORK
TITLE =WW: Folge 2 Tx M6 Spindel belegt / Auftrag 3

      U     #Vorbedingung_AF2;
      U     "DB_WW".WW_gestartet; // STARTEN VON WZW-ABLAUF
      UN    "DB_WW".WW_SEMA_Folgen; // SEMA ABLAUFFOLGEN
      S     "DB_WW".WW_SEMA_Folgen; // SEMA ABLAUFFOLGEN
      S     "DB_WW".WW_T_Auftrag_3; // AUFTRAG3 ABLEGEN II ->Z-HUB EINGEFAHREN
      S     "DB_WW".WW_T_Folge_2; // ABLAUFFOLGE 2
      S     "DB_WW".WW_Hschritt_1; // HILFSSCHRITT1

NETWORK
TITLE =WW: Folge 2 Freigabe fahre ins Magazin

      U     "DB_WW".WW_T_Auftrag_3; // AUFTRAG3 ABLEGEN II ->Z-HUB EINGEFAHREN
      U     "DB_WW".WW_T_Folge_2; // ABLAUFFOLGE 2
      U     "DB_WZV".Mag1_inPos_WST;
      U(    ;
      O     "I_WW_MagPlatz_frei"; // WZ in Wechselposition (Magazinplatz frei)
      O     #IB_MagKontr_aus; // Kontrolle Magazinplatz ausblenden
      )     ;
      S     "DB_WW".WW_Frg_ins_Mag; // FREIGABE FAHRE INS MAGAZIN

NETWORK
TITLE =WW: Folge 2 HILFSSCHRITT2
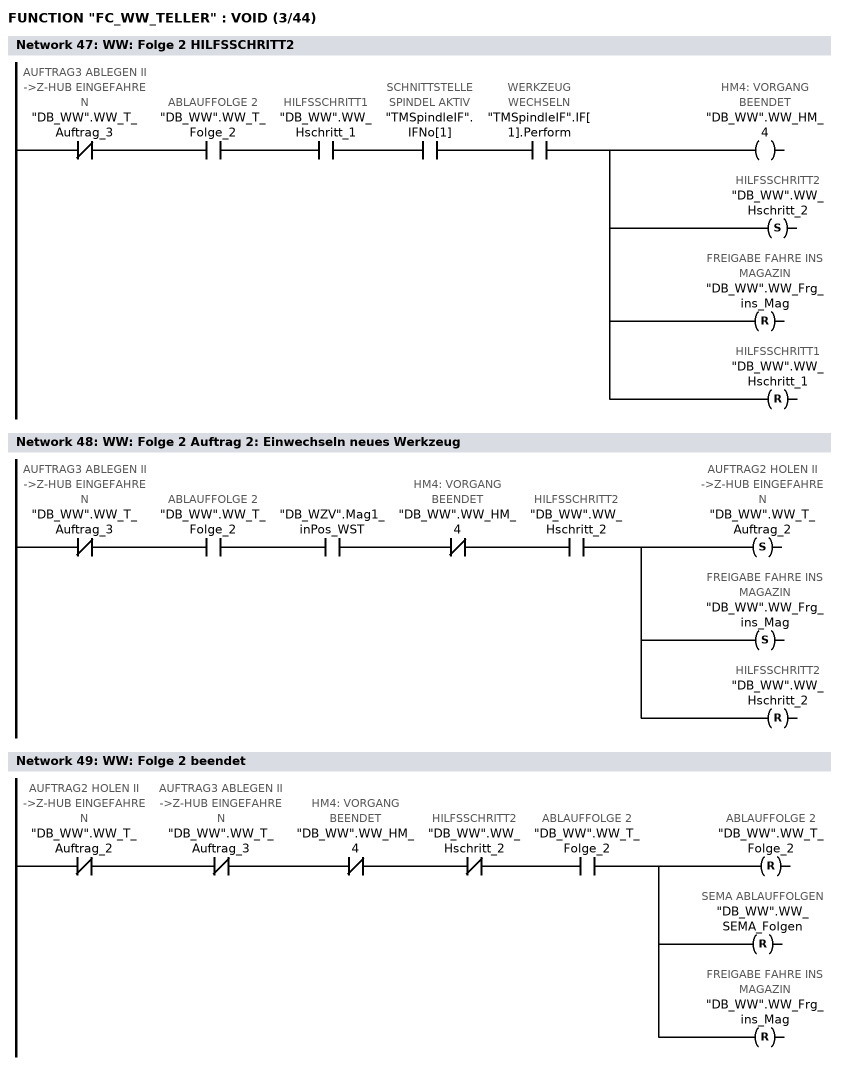

      UN    "DB_WW".WW_T_Auftrag_3; // AUFTRAG3 ABLEGEN II ->Z-HUB EINGEFAHREN
      U     "DB_WW".WW_T_Folge_2; // ABLAUFFOLGE 2
      U     "DB_WW".WW_Hschritt_1; // HILFSSCHRITT1
      U     "TMSpindleIF".IFNo[1]; // SCHNITTSTELLE SPINDEL AKTIV
      U     "TMSpindleIF".IF[1].Perform; // WERKZEUG WECHSELN
      =     "DB_WW".WW_HM_4; // HM4: VORGANG BEENDET
      S     "DB_WW".WW_Hschritt_2; // HILFSSCHRITT2
      R     "DB_WW".WW_Frg_ins_Mag; // FREIGABE FAHRE INS MAGAZIN
      R     "DB_WW".WW_Hschritt_1; // HILFSSCHRITT1

NETWORK
TITLE =WW: Folge 2 Auftrag 2: Einwechseln neues Werkzeug

      UN    "DB_WW".WW_T_Auftrag_3; // AUFTRAG3 ABLEGEN II ->Z-HUB EINGEFAHREN
      U     "DB_WW".WW_T_Folge_2; // ABLAUFFOLGE 2
      U     "DB_WZV".Mag1_inPos_WST;
      UN    "DB_WW".WW_HM_4; // HM4: VORGANG BEENDET
      U     "DB_WW".WW_Hschritt_2; // HILFSSCHRITT2
      S     "DB_WW".WW_T_Auftrag_2; // AUFTRAG2 HOLEN II ->Z-HUB EINGEFAHREN
      S     "DB_WW".WW_Frg_ins_Mag; // FREIGABE FAHRE INS MAGAZIN
      R     "DB_WW".WW_Hschritt_2; // HILFSSCHRITT2

NETWORK
TITLE =WW: Folge 2 beendet

      UN    "DB_WW".WW_T_Auftrag_2; // AUFTRAG2 HOLEN II ->Z-HUB EINGEFAHREN
      UN    "DB_WW".WW_T_Auftrag_3; // AUFTRAG3 ABLEGEN II ->Z-HUB EINGEFAHREN
      UN    "DB_WW".WW_HM_4; // HM4: VORGANG BEENDET
      UN    "DB_WW".WW_Hschritt_2; // HILFSSCHRITT2
      U     "DB_WW".WW_T_Folge_2; // ABLAUFFOLGE 2
      R     "DB_WW".WW_T_Folge_2; // ABLAUFFOLGE 2
      R     "DB_WW".WW_SEMA_Folgen; // SEMA ABLAUFFOLGEN
      R     "DB_WW".WW_Frg_ins_Mag; // FREIGABE FAHRE INS MAGAZIN

NETWORK
TITLE =WW: Folge 3 T0 M6 Spindel belegt / Auftrag 3
//3.AUFTRAGSFOLGE: SPINDEL BELEGT UND T0 PROGRAMMIERT
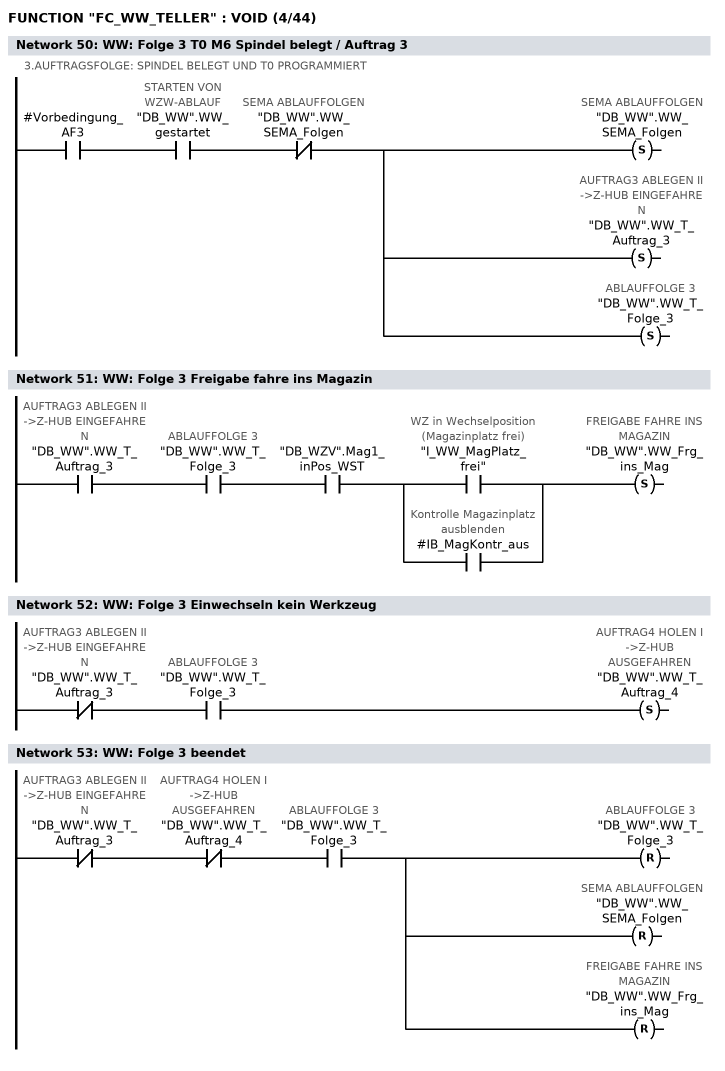
      U     #Vorbedingung_AF3;
      U     "DB_WW".WW_gestartet; // STARTEN VON WZW-ABLAUF
      UN    "DB_WW".WW_SEMA_Folgen; // SEMA ABLAUFFOLGEN
      S     "DB_WW".WW_SEMA_Folgen; // SEMA ABLAUFFOLGEN
      S     "DB_WW".WW_T_Auftrag_3; // AUFTRAG3 ABLEGEN II ->Z-HUB EINGEFAHREN
      S     "DB_WW".WW_T_Folge_3; // ABLAUFFOLGE 3

NETWORK
TITLE =WW: Folge 3 Freigabe fahre ins Magazin

      U     "DB_WW".WW_T_Auftrag_3; // AUFTRAG3 ABLEGEN II ->Z-HUB EINGEFAHREN
      U     "DB_WW".WW_T_Folge_3; // ABLAUFFOLGE 3
      U     "DB_WZV".Mag1_inPos_WST;
      U(    ;
      O     "I_WW_MagPlatz_frei"; // WZ in Wechselposition (Magazinplatz frei)
      O     #IB_MagKontr_aus; // Kontrolle Magazinplatz ausblenden
      )     ;
      S     "DB_WW".WW_Frg_ins_Mag; // FREIGABE FAHRE INS MAGAZIN

NETWORK
TITLE =WW: Folge 3 Einwechseln kein Werkzeug

      UN    "DB_WW".WW_T_Auftrag_3; // AUFTRAG3 ABLEGEN II ->Z-HUB EINGEFAHREN
      U     "DB_WW".WW_T_Folge_3; // ABLAUFFOLGE 3
      S     "DB_WW".WW_T_Auftrag_4; // AUFTRAG4 HOLEN I ->Z-HUB AUSGEFAHREN

NETWORK
TITLE =WW: Folge 3 beendet

      UN    "DB_WW".WW_T_Auftrag_3; // AUFTRAG3 ABLEGEN II ->Z-HUB EINGEFAHREN
      UN    "DB_WW".WW_T_Auftrag_4; // AUFTRAG4 HOLEN I ->Z-HUB AUSGEFAHREN
      U     "DB_WW".WW_T_Folge_3; // ABLAUFFOLGE 3
      R     "DB_WW".WW_T_Folge_3; // ABLAUFFOLGE 3
      R     "DB_WW".WW_SEMA_Folgen; // SEMA ABLAUFFOLGEN
      R     "DB_WW".WW_Frg_ins_Mag; // FREIGABE FAHRE INS MAGAZIN

NETWORK
TITLE =WW: ABBRUCH -> FREIFAHREN
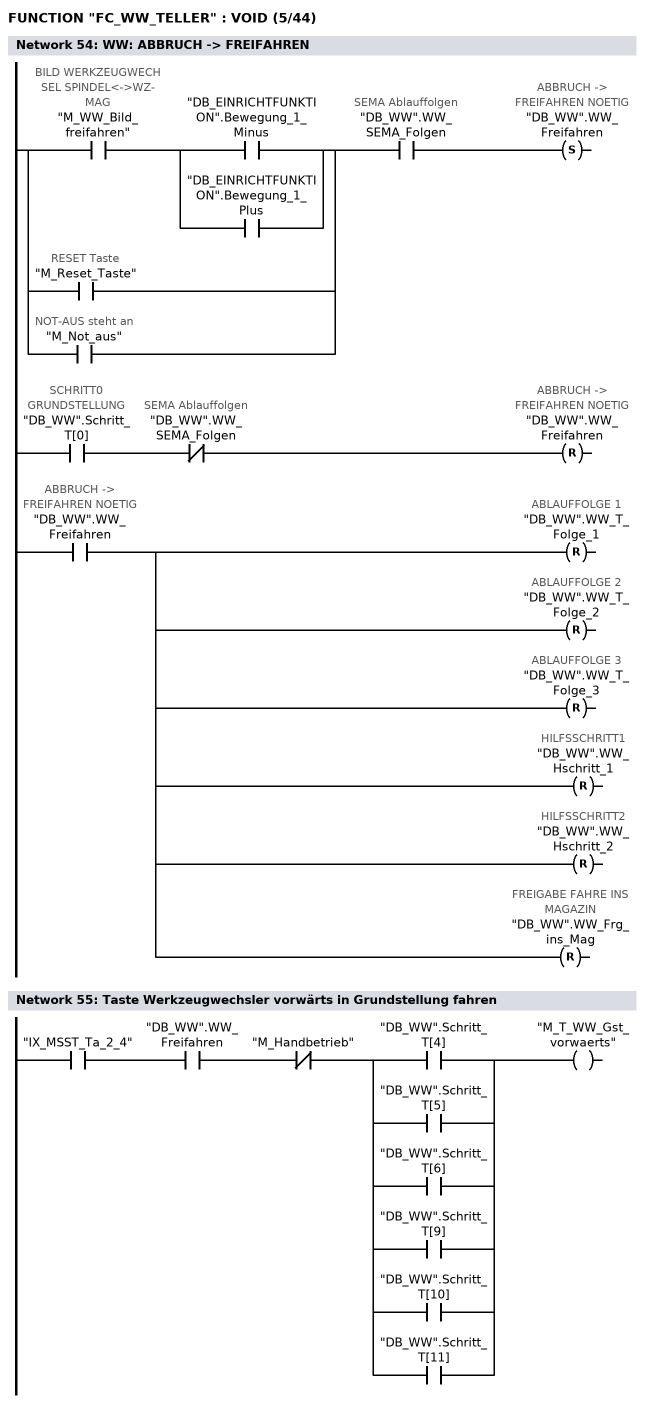

      U(    ;
      U     "M_WW_Bild_freifahren"; // BILD WERKZEUGWECHSEL SPINDEL<->WZ-MAG
      U(    ;
      O     "DB_EINRICHTFUNKTION".Bewegung_1_Minus;
      O     "DB_EINRICHTFUNKTION".Bewegung_1_Plus;
      )     ;
      O     "M_Reset_Taste"; // RESET Taste
      O     "M_Not_aus"; // NOT-AUS steht an
      )     ;
      U     "DB_WW".WW_SEMA_Folgen; // SEMA Ablauffolgen
      S     "DB_WW".WW_Freifahren; // ABBRUCH -> FREIFAHREN NOETIG

      U     "DB_WW".Schritt_T[0]; // SCHRITT0 GRUNDSTELLUNG
      UN    "DB_WW".WW_SEMA_Folgen; // SEMA Ablauffolgen
      R     "DB_WW".WW_Freifahren; // ABBRUCH -> FREIFAHREN NOETIG

      U     "DB_WW".WW_Freifahren; // ABBRUCH -> FREIFAHREN NOETIG
      R     "DB_WW".WW_T_Folge_1; // ABLAUFFOLGE 1
      R     "DB_WW".WW_T_Folge_2; // ABLAUFFOLGE 2
      R     "DB_WW".WW_T_Folge_3; // ABLAUFFOLGE 3
      R     "DB_WW".WW_Hschritt_1; // HILFSSCHRITT1
      R     "DB_WW".WW_Hschritt_2; // HILFSSCHRITT2
      R     "DB_WW".WW_Frg_ins_Mag; // FREIGABE FAHRE INS MAGAZIN

NETWORK
TITLE =Taste Werkzeugwechsler vorwärts in Grundstellung fahren

      U     "IX_MSST_Ta_2_4";
      U     "DB_WW".WW_Freifahren;
      UN    "M_Handbetrieb";
      U(    ;
      O     "DB_WW".Schritt_T[4];
      O     "DB_WW".Schritt_T[5];
      O     "DB_WW".Schritt_T[6];
      O     "DB_WW".Schritt_T[9];
      O     "DB_WW".Schritt_T[10];
      O     "DB_WW".Schritt_T[11];
      )     ;
      =     "M_T_WW_Gst_vorwaerts";


NETWORK
TITLE =Taste Werkzeugwechsler rückwärts in Grundstellung fahren
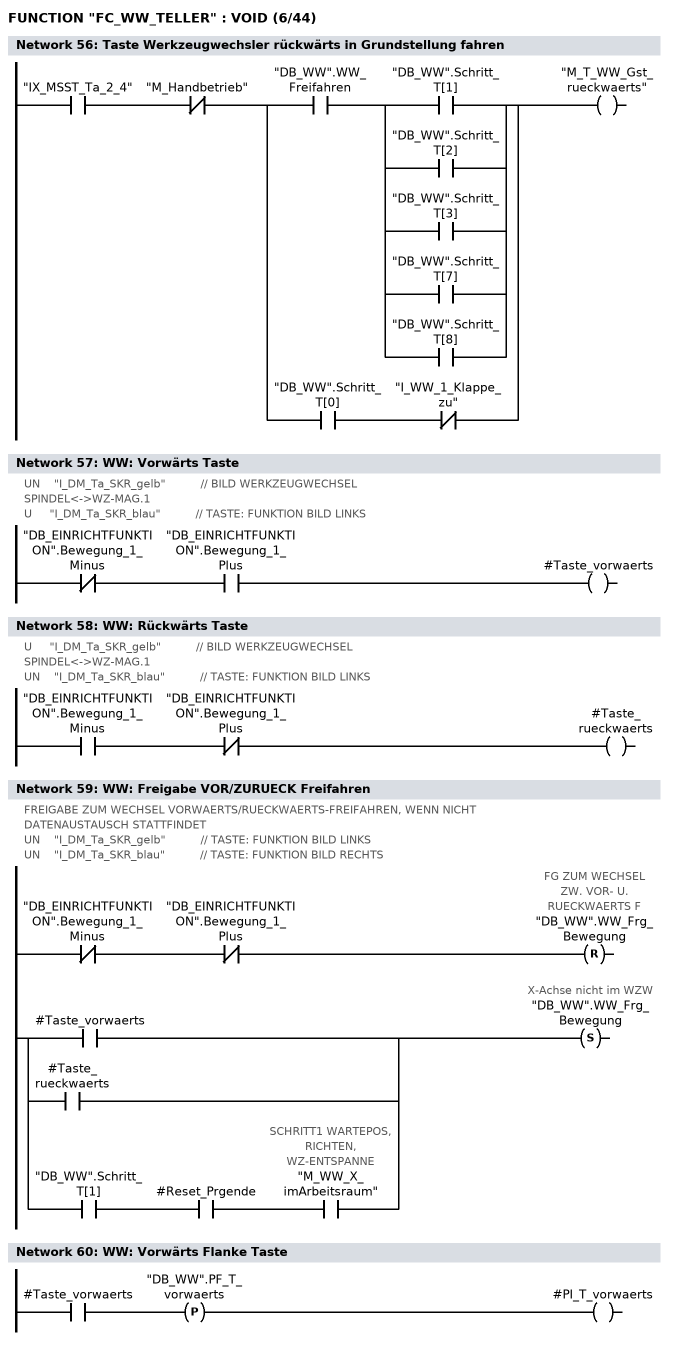

      U     "IX_MSST_Ta_2_4";
      UN    "M_Handbetrieb";
      U(    ;
      U     "DB_WW".WW_Freifahren;
      U(    ;
      O     "DB_WW".Schritt_T[1];
      O     "DB_WW".Schritt_T[2];
      O     "DB_WW".Schritt_T[3];
      O     "DB_WW".Schritt_T[7];
      O     "DB_WW".Schritt_T[8];
      )     ;
      O     ;
      U     "DB_WW".Schritt_T[0];
      UN    "I_WW_1_Klappe_zu";
      )     ;
      =     "M_T_WW_Gst_rueckwaerts";

NETWORK
TITLE =WW: Vorwärts Taste
//      UN    "I_DM_Ta_SKR_gelb"          // BILD WERKZEUGWECHSEL
//SPINDEL<->WZ-MAG.1
//      U     "I_DM_Ta_SKR_blau"          // TASTE: FUNKTION BILD LINKS
      UN    "DB_EINRICHTFUNKTION".Bewegung_1_Minus;
      U     "DB_EINRICHTFUNKTION".Bewegung_1_Plus;
      =     #Taste_vorwaerts;

NETWORK
TITLE =WW: Rückwärts Taste
//      U     "I_DM_Ta_SKR_gelb"          // BILD WERKZEUGWECHSEL
//SPINDEL<->WZ-MAG.1
//      UN    "I_DM_Ta_SKR_blau"          // TASTE: FUNKTION BILD LINKS
      U     "DB_EINRICHTFUNKTION".Bewegung_1_Minus;
      UN    "DB_EINRICHTFUNKTION".Bewegung_1_Plus;
      =     #Taste_rueckwaerts;

NETWORK
TITLE =WW: Freigabe VOR/ZURUECK Freifahren
// FREIGABE ZUM WECHSEL VORWAERTS/RUECKWAERTS-FREIFAHREN, WENN NICHT
// DATENAUSTAUSCH STATTFINDET
//      UN    "I_DM_Ta_SKR_gelb"          // TASTE: FUNKTION BILD LINKS
//      UN    "I_DM_Ta_SKR_blau"          // TASTE: FUNKTION BILD RECHTS
      UN    "DB_EINRICHTFUNKTION".Bewegung_1_Minus;
      UN    "DB_EINRICHTFUNKTION".Bewegung_1_Plus;
      R     "DB_WW".WW_Frg_Bewegung; // FG ZUM WECHSEL ZW. VOR- U. RUECKWAERTS F

      U(    ;
      O     #Taste_vorwaerts;
      O     #Taste_rueckwaerts;
      O     ; // TASTE: FUNKTION BILD LINKS
      U     "DB_WW".Schritt_T[1];
      U     #Reset_Prgende;
      U     "M_WW_X_imArbeitsraum"; // SCHRITT1 WARTEPOS, RICHTEN, WZ-ENTSPANNE
      )     ; // RESET KANAL 1
      S     "DB_WW".WW_Frg_Bewegung; // X-Achse nicht im WZW
      NOP   0;
NETWORK
TITLE =WW: Vorwärts Flanke Taste

      U     #Taste_vorwaerts;
      FP    "DB_WW".PF_T_vorwaerts;
      =     #PI_T_vorwaerts;

NETWORK
TITLE =WW: Vorwärts Bewegung
// ZUR STEUERUNG DER SCHRITTKETTE MUSS DIE RICHTUNG, WELCHE DIE SCHRITT-
// KETTE MACHT FESTGELEGT WERDEN
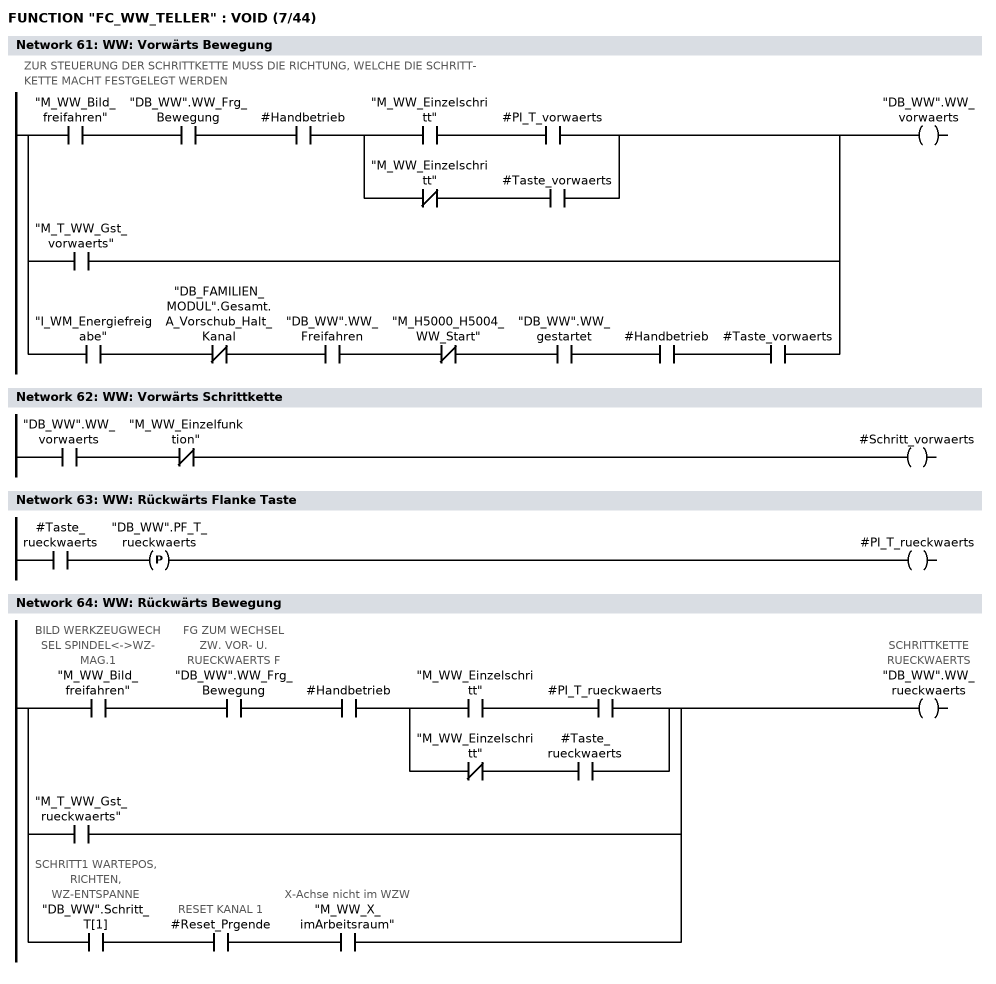
      U     "M_WW_Bild_freifahren";
      U     "DB_WW".WW_Frg_Bewegung;
      U     #Handbetrieb;
      U(    ;
      U     "M_WW_Einzelschritt";
      U     #PI_T_vorwaerts;
      O     ;
      UN    "M_WW_Einzelschritt";
      U     #Taste_vorwaerts;
      )     ;
      O     "M_T_WW_Gst_vorwaerts";
      O     ;
      U     "I_WM_Energiefreigabe";
      UN    "DB_FAMILIEN_MODUL".Gesamt.A_Vorschub_Halt_Kanal;
      U     "DB_WW".WW_Freifahren;
      UN    "M_H5000_H5004_WW_Start";
      U     "DB_WW".WW_gestartet;
      U     #Handbetrieb;
      U     #Taste_vorwaerts;
      =     "DB_WW".WW_vorwaerts;
NETWORK
TITLE =WW: Vorwärts Schrittkette

      U     "DB_WW".WW_vorwaerts;
      UN    "M_WW_Einzelfunktion";
      =     #Schritt_vorwaerts;

NETWORK
TITLE =WW: Rückwärts Flanke Taste

      U     #Taste_rueckwaerts;
      FP    "DB_WW".PF_T_rueckwaerts;
      =     #PI_T_rueckwaerts;

NETWORK
TITLE =WW: Rückwärts Bewegung

      U     "M_WW_Bild_freifahren"; // BILD WERKZEUGWECHSEL SPINDEL<->WZ-MAG.1
      U     "DB_WW".WW_Frg_Bewegung; // FG ZUM WECHSEL ZW. VOR- U. RUECKWAERTS F
      U     #Handbetrieb;
      U(    ;
      U     "M_WW_Einzelschritt";
      U     #PI_T_rueckwaerts;
      O     ;
      UN    "M_WW_Einzelschritt";
      U     #Taste_rueckwaerts;
      )     ;
      O     "M_T_WW_Gst_rueckwaerts";
      O     ;
      U     "DB_WW".Schritt_T[1]; // SCHRITT1 WARTEPOS, RICHTEN, WZ-ENTSPANNE
      U     #Reset_Prgende; // RESET KANAL 1
      U     "M_WW_X_imArbeitsraum"; // X-Achse nicht im WZW
      =     "DB_WW".WW_rueckwaerts; // SCHRITTKETTE RUECKWAERTS

NETWORK
TITLE =WW: Rückwärts gespeichert
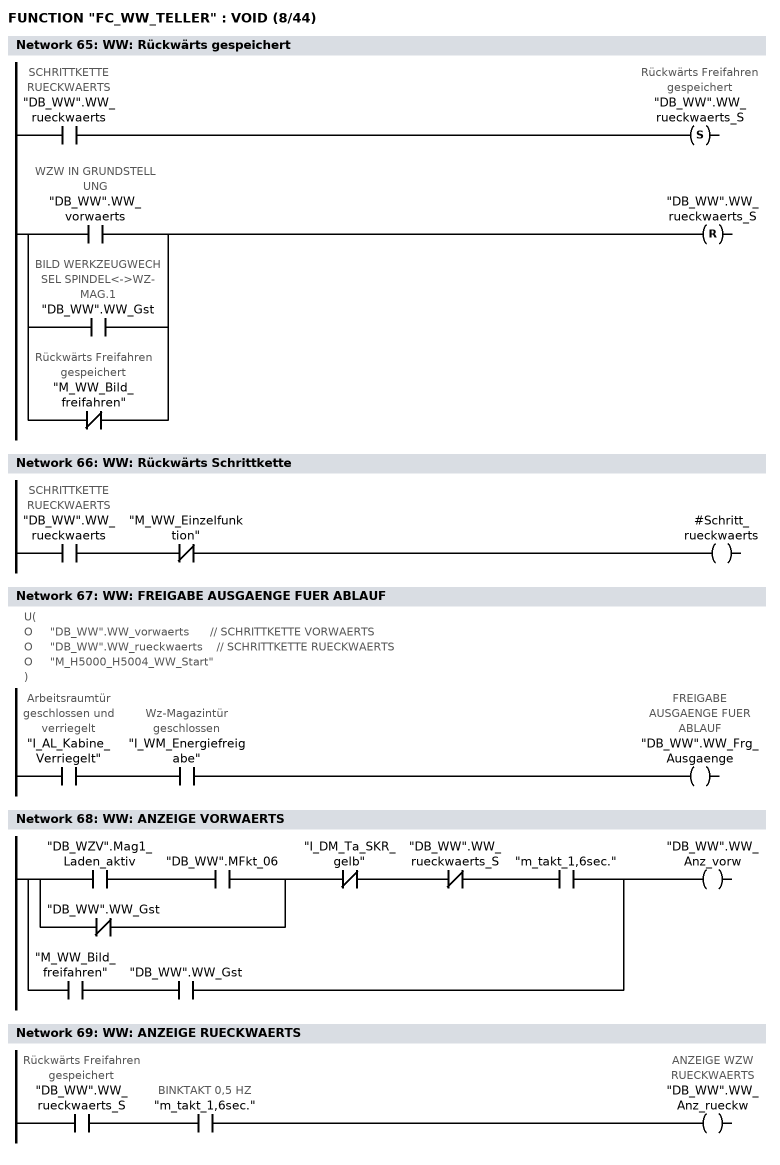

      U     "DB_WW".WW_rueckwaerts; // SCHRITTKETTE RUECKWAERTS
      S     "DB_WW".WW_rueckwaerts_S; // Rückwärts Freifahren gespeichert


      U(    ; // SCHRITTKETTE VORWAERTS
      O     "DB_WW".WW_vorwaerts; // WZW IN GRUNDSTELLUNG
      O     "DB_WW".WW_Gst; // BILD WERKZEUGWECHSEL SPINDEL<->WZ-MAG.1
      ON    "M_WW_Bild_freifahren"; // Rückwärts Freifahren gespeichert
      )     ;

      R     "DB_WW".WW_rueckwaerts_S;
      NOP   0;
NETWORK
TITLE =WW: Rückwärts Schrittkette

      U     "DB_WW".WW_rueckwaerts; // SCHRITTKETTE RUECKWAERTS
      UN    "M_WW_Einzelfunktion";
      =     #Schritt_rueckwaerts;

NETWORK
TITLE =WW: FREIGABE AUSGAENGE FUER ABLAUF
//      U(
//      O     "DB_WW".WW_vorwaerts      // SCHRITTKETTE VORWAERTS
//      O     "DB_WW".WW_rueckwaerts    // SCHRITTKETTE RUECKWAERTS
//      O     "M_H5000_H5004_WW_Start"
//      )
      U     "I_AL_Kabine_Verriegelt"; // Arbeitsraumtür geschlossen und verriegelt
      U     "I_WM_Energiefreigabe"; // Wz-Magazintür geschlossen
      =     "DB_WW".WW_Frg_Ausgaenge; // FREIGABE AUSGAENGE FUER ABLAUF

NETWORK
TITLE =WW: ANZEIGE VORWAERTS

      U(    ;
      U     "DB_WZV".Mag1_Laden_aktiv;
      U     "DB_WW".MFkt_06;
      ON    "DB_WW".WW_Gst;
      )     ;
      UN    "I_DM_Ta_SKR_gelb";
      UN    "DB_WW".WW_rueckwaerts_S;
      U     "m_takt_1,6sec.";
      O     ;
      U     "M_WW_Bild_freifahren";
      U     "DB_WW".WW_Gst;
      =     "DB_WW".WW_Anz_vorw;
NETWORK
TITLE =WW: ANZEIGE RUECKWAERTS

      U     "DB_WW".WW_rueckwaerts_S; // Rückwärts Freifahren gespeichert
      U     "m_takt_1,6sec."; // BINKTAKT 0,5 HZ
      =     "DB_WW".WW_Anz_rueckw; // ANZEIGE WZW RUECKWAERTS

NETWORK
TITLE =WW: Semifunktion Ansteuerung Anzeige Werkzeugwechsler
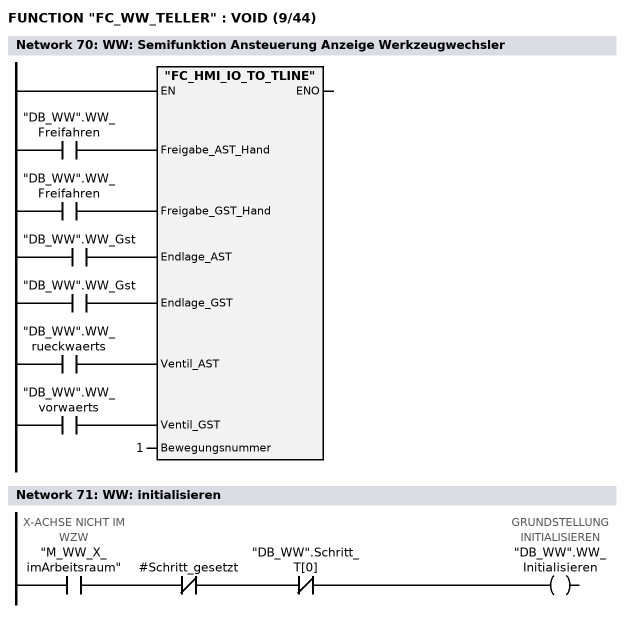

      U     "DB_WW".WW_Freifahren;
      =     L     24.0;
      BLD   103;
      U     "DB_WW".WW_Freifahren;
      =     L     24.1;
      BLD   103;
      U     "DB_WW".WW_Gst;
      =     L     24.2;
      BLD   103;
      U     "DB_WW".WW_Gst;
      =     L     24.3;
      BLD   103;
      U     "DB_WW".WW_rueckwaerts;
      =     L     24.4;
      BLD   103;
      U     "DB_WW".WW_vorwaerts;
      =     L     24.5;
      BLD   103;
      CALL "FC_HMI_IO_TO_TLINE" (
           Freigabe_AST_Hand        := L     24.0,
           Freigabe_GST_Hand        := L     24.1,
           Endlage_AST              := L     24.2,
           Endlage_GST              := L     24.3,
           Ventil_AST               := L     24.4,
           Ventil_GST               := L     24.5,
           Bewegungsnummer          := 1);
      NOP   0;
NETWORK
TITLE =WW: initialisieren

      U     "M_WW_X_imArbeitsraum"; // X-ACHSE NICHT IM WZW
      UN    #Schritt_gesetzt;
      UN    "DB_WW".Schritt_T[0];
      =     "DB_WW".WW_Initialisieren; // GRUNDSTELLUNG INITIALISIEREN

NETWORK
TITLE =WW: SCHRITT_0 GRUNDSTELLUNG
// DER SCHRITT0 IST DER SCHRITT, WELCHER NACH JEDEM WZ-WECHSEL ANGELAUFEN
// WERDEN MUSS.
//
// X-ACHSE NICHT IM WECHSLER
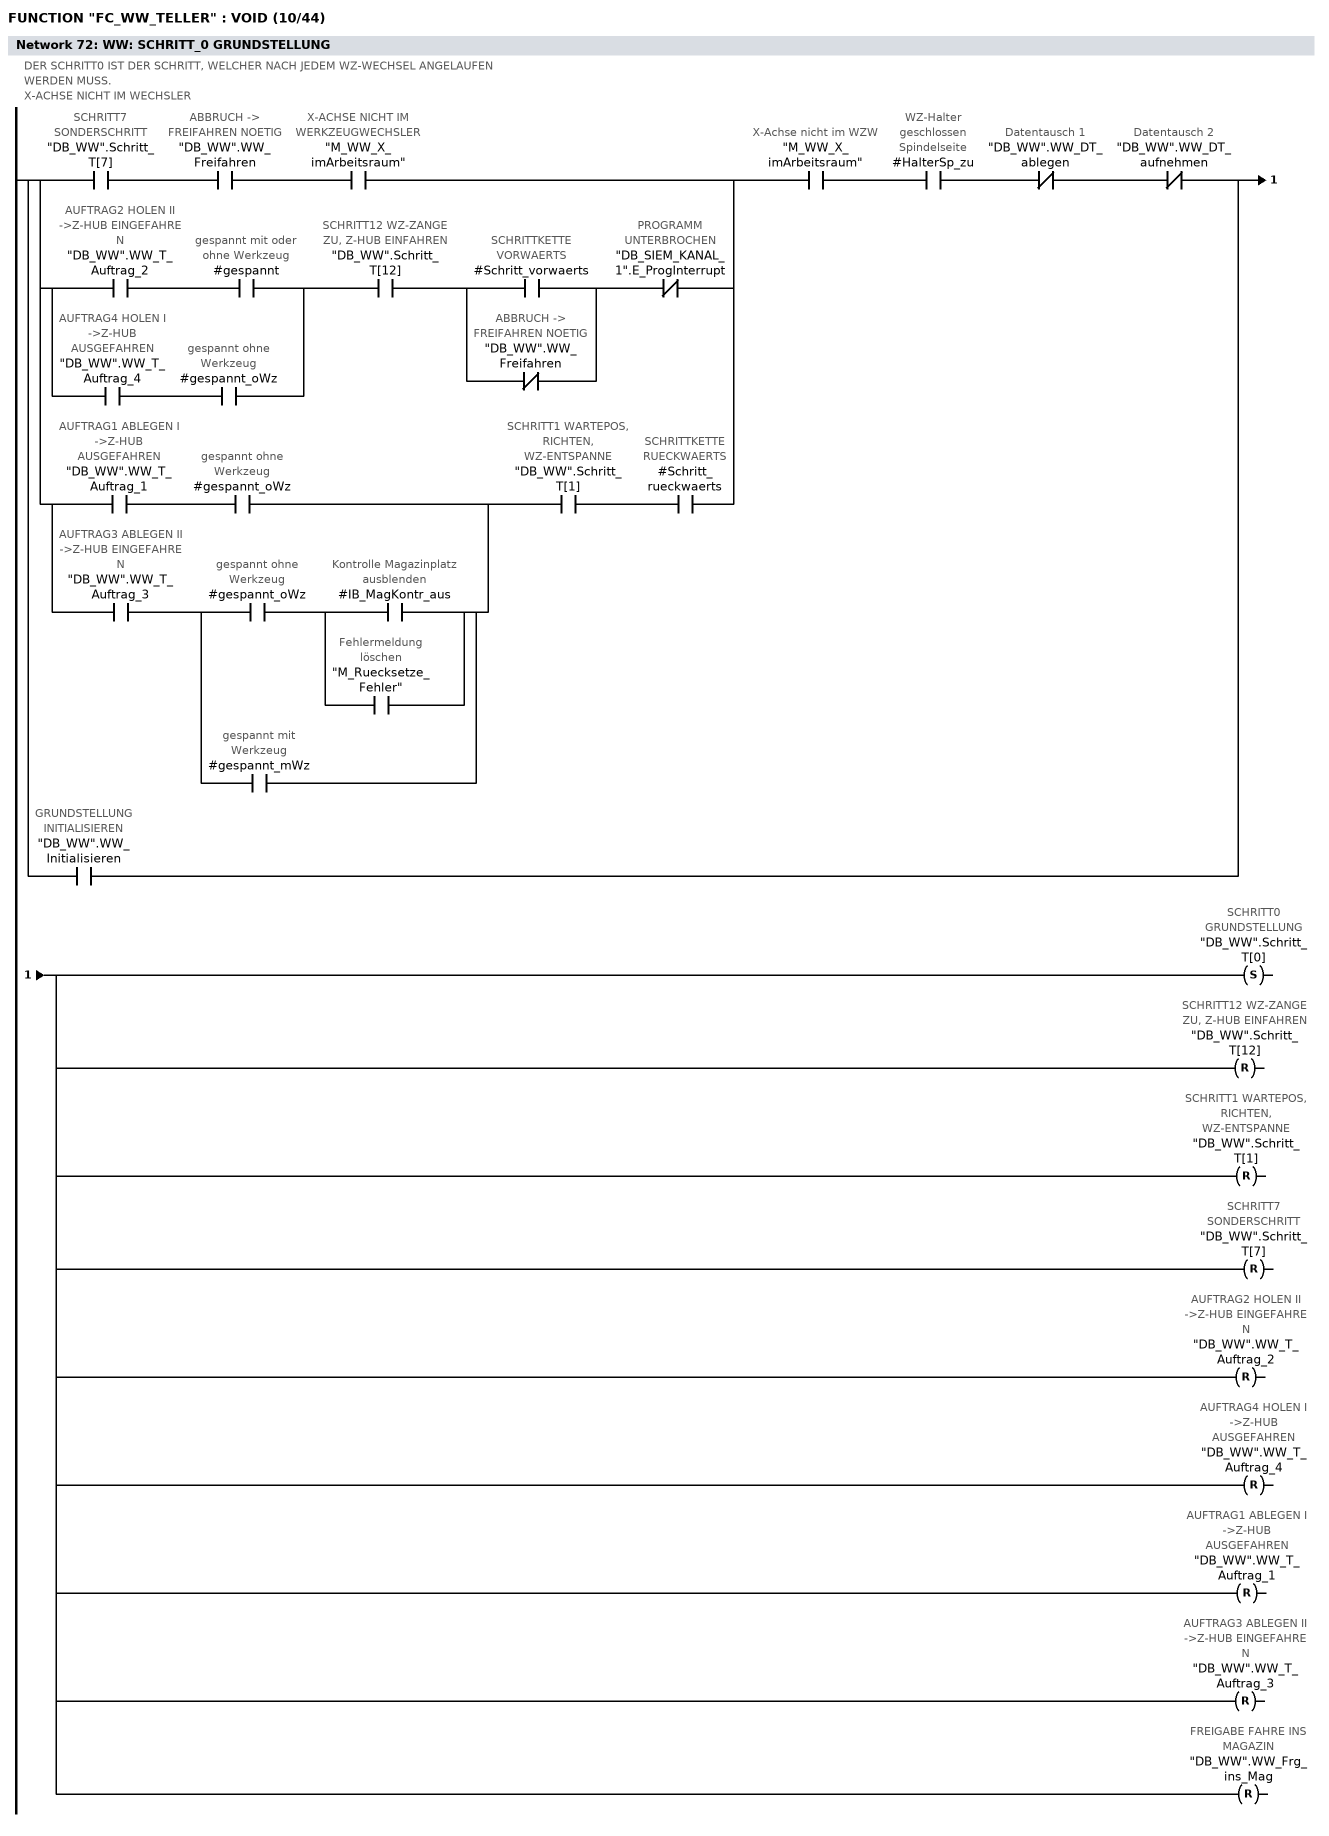
      U(    ;
      U     "DB_WW".Schritt_T[7]; // SCHRITT7 SONDERSCHRITT
      U     "DB_WW".WW_Freifahren; // ABBRUCH -> FREIFAHREN NOETIG
      U     "M_WW_X_imArbeitsraum"; // X-ACHSE NICHT IM WERKZEUGWECHSLER

      O     ;
      U(    ;
      U     "DB_WW".WW_T_Auftrag_2; // AUFTRAG2 HOLEN II ->Z-HUB EINGEFAHREN
      U     #gespannt; // gespannt mit oder ohne Werkzeug
      O     ;
      U     "DB_WW".WW_T_Auftrag_4; // AUFTRAG4 HOLEN I ->Z-HUB AUSGEFAHREN
      U     #gespannt_oWz; // gespannt ohne Werkzeug
      )     ;
      U     "DB_WW".Schritt_T[12]; // SCHRITT12 WZ-ZANGE ZU, Z-HUB EINFAHREN
      U(    ;
      O     #Schritt_vorwaerts; // SCHRITTKETTE VORWAERTS
      ON    "DB_WW".WW_Freifahren; // ABBRUCH -> FREIFAHREN NOETIG
      )     ;
      UN    "DB_SIEM_KANAL_1".E_ProgInterrupt; // PROGRAMM UNTERBROCHEN

      O     ;
      U(    ;
      U     "DB_WW".WW_T_Auftrag_1; // AUFTRAG1 ABLEGEN I ->Z-HUB AUSGEFAHREN
      U     #gespannt_oWz; // gespannt ohne Werkzeug
      O     ;
      U     "DB_WW".WW_T_Auftrag_3; // AUFTRAG3 ABLEGEN II ->Z-HUB EINGEFAHREN
      U(    ;
      U     #gespannt_oWz; // gespannt ohne Werkzeug
      U(    ;
      O     #IB_MagKontr_aus; // Kontrolle Magazinplatz ausblenden
      O     "M_Ruecksetze_Fehler"; // Fehlermeldung löschen
      )     ;
      O     #gespannt_mWz; // gespannt mit Werkzeug
      )     ;
      )     ;
      U     "DB_WW".Schritt_T[1]; // SCHRITT1 WARTEPOS, RICHTEN, WZ-ENTSPANNE
      U     #Schritt_rueckwaerts; // SCHRITTKETTE RUECKWAERTS

      )     ;
      U     "M_WW_X_imArbeitsraum"; // X-Achse nicht im WZW
      U     #HalterSp_zu; // WZ-Halter geschlossen Spindelseite
      UN    "DB_WW".WW_DT_ablegen; // Datentausch 1
      UN    "DB_WW".WW_DT_aufnehmen; // Datentausch 2

      O     "DB_WW".WW_Initialisieren; // GRUNDSTELLUNG INITIALISIEREN

      S     "DB_WW".Schritt_T[0]; // SCHRITT0 GRUNDSTELLUNG
      R     "DB_WW".Schritt_T[12]; // SCHRITT12 WZ-ZANGE ZU, Z-HUB EINFAHREN
      R     "DB_WW".Schritt_T[1]; // SCHRITT1 WARTEPOS, RICHTEN, WZ-ENTSPANNE
      R     "DB_WW".Schritt_T[7]; // SCHRITT7 SONDERSCHRITT
      R     "DB_WW".WW_T_Auftrag_2; // AUFTRAG2 HOLEN II ->Z-HUB EINGEFAHREN
      R     "DB_WW".WW_T_Auftrag_4; // AUFTRAG4 HOLEN I ->Z-HUB AUSGEFAHREN
      R     "DB_WW".WW_T_Auftrag_1; // AUFTRAG1 ABLEGEN I ->Z-HUB AUSGEFAHREN
      R     "DB_WW".WW_T_Auftrag_3; // AUFTRAG3 ABLEGEN II ->Z-HUB EINGEFAHREN
      R     "DB_WW".WW_Frg_ins_Mag; // FREIGABE FAHRE INS MAGAZIN

NETWORK
TITLE =WW: GRUNDSTELLUNG MELDEN
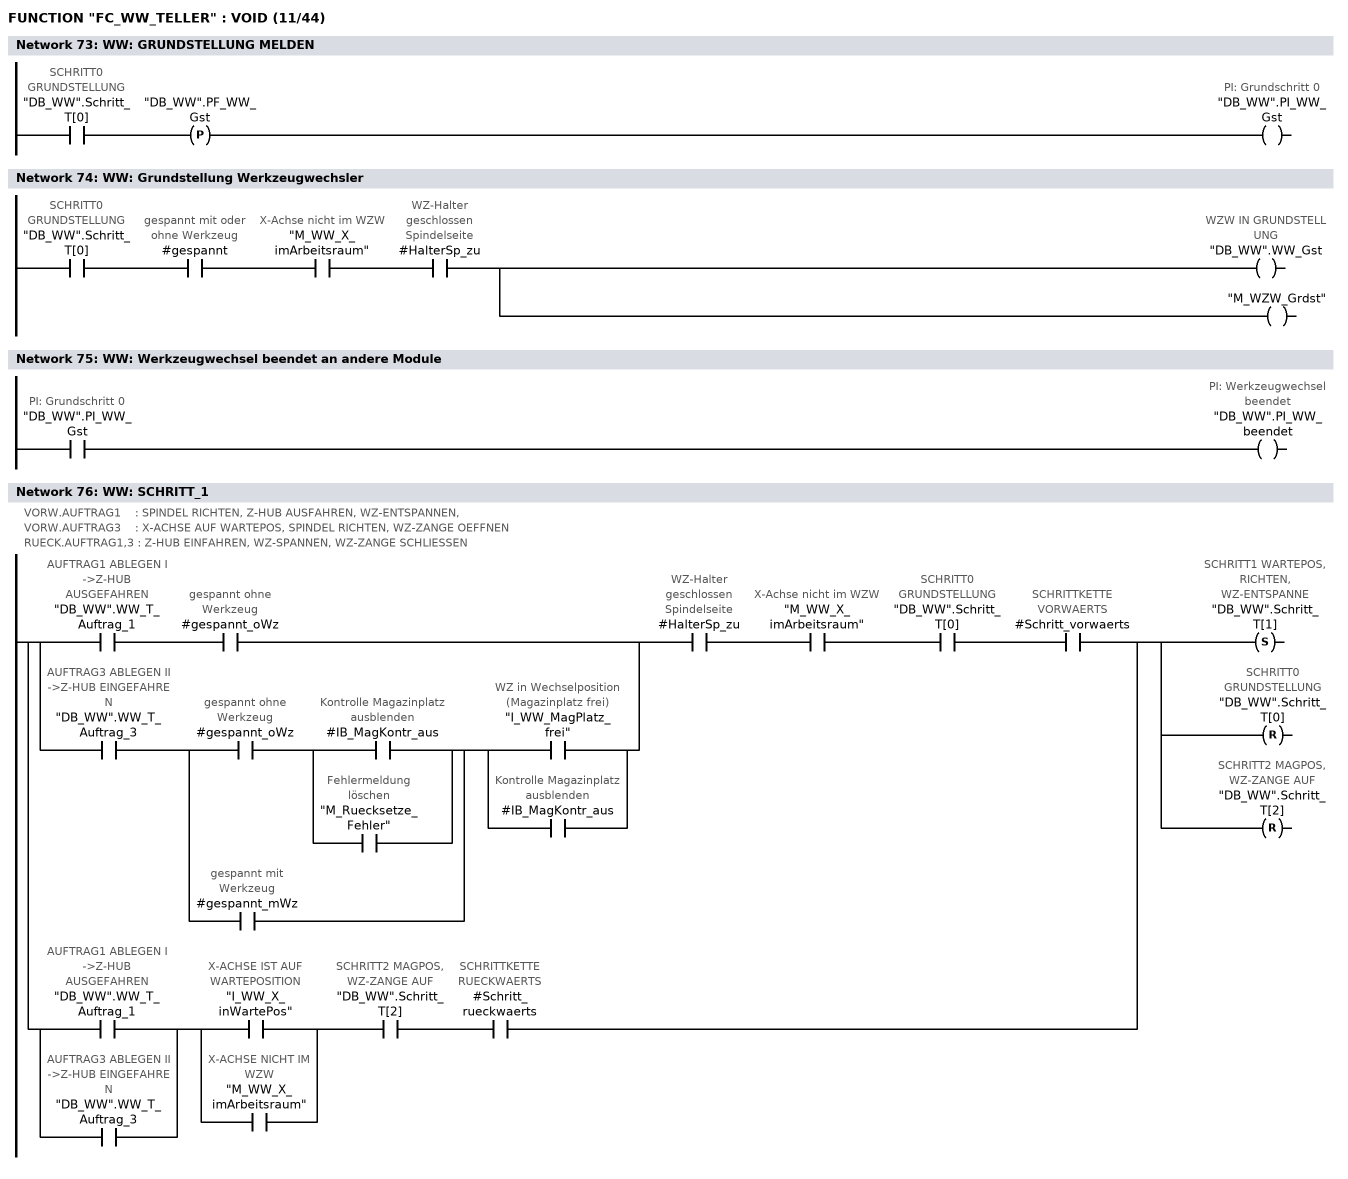

      U     "DB_WW".Schritt_T[0]; // SCHRITT0 GRUNDSTELLUNG
      FP    "DB_WW".PF_WW_Gst; // PF: Werkzeugwechsel in Schritt 0
      =     "DB_WW".PI_WW_Gst; // PI: Grundschritt 0

NETWORK
TITLE =WW: Grundstellung Werkzeugwechsler

      U     "DB_WW".Schritt_T[0]; // SCHRITT0 GRUNDSTELLUNG
      U     #gespannt; // gespannt mit oder ohne Werkzeug
      U     "M_WW_X_imArbeitsraum"; // X-Achse nicht im WZW
      U     #HalterSp_zu; // WZ-Halter geschlossen Spindelseite
      =     "DB_WW".WW_Gst; // WZW IN GRUNDSTELLUNG
      =     "M_WZW_Grdst";
NETWORK
TITLE =WW: Werkzeugwechsel beendet an andere Module

      U     "DB_WW".PI_WW_Gst; // PI: Grundschritt 0
      =     "DB_WW".PI_WW_beendet; // PI: Werkzeugwechsel beendet

NETWORK
TITLE =WW: SCHRITT_1
// VORW.AUFTRAG1    : SPINDEL RICHTEN, Z-HUB AUSFAHREN, WZ-ENTSPANNEN,
// VORW.AUFTRAG3    : X-ACHSE AUF WARTEPOS, SPINDEL RICHTEN, WZ-ZANGE OEFFNEN
// RUECK.AUFTRAG1,3 : Z-HUB EINFAHREN, WZ-SPANNEN, WZ-ZANGE SCHLIESSEN
      U(    ;
      U     "DB_WW".WW_T_Auftrag_1; // AUFTRAG1 ABLEGEN I ->Z-HUB AUSGEFAHREN
      U     #gespannt_oWz; // gespannt ohne Werkzeug
      O     ;
      U     "DB_WW".WW_T_Auftrag_3; // AUFTRAG3 ABLEGEN II ->Z-HUB EINGEFAHREN
      U(    ;
      U     #gespannt_oWz; // gespannt ohne Werkzeug
      U(    ;
      O     #IB_MagKontr_aus; // Kontrolle Magazinplatz ausblenden
      O     "M_Ruecksetze_Fehler"; // Fehlermeldung löschen
      )     ;
      O     #gespannt_mWz; // gespannt mit Werkzeug
      )     ;
      U(    ;
      O     "I_WW_MagPlatz_frei"; // WZ in Wechselposition (Magazinplatz frei)
      O     #IB_MagKontr_aus; // Kontrolle Magazinplatz ausblenden
      )     ;
      )     ;
      U     #HalterSp_zu; // WZ-Halter geschlossen Spindelseite
      U     "M_WW_X_imArbeitsraum"; // X-Achse nicht im WZW
      U     "DB_WW".Schritt_T[0]; // SCHRITT0 GRUNDSTELLUNG
      U     #Schritt_vorwaerts; // SCHRITTKETTE VORWAERTS

      O     ;
      U(    ;
      O     "DB_WW".WW_T_Auftrag_1; // AUFTRAG1 ABLEGEN I ->Z-HUB AUSGEFAHREN
      O     "DB_WW".WW_T_Auftrag_3; // AUFTRAG3 ABLEGEN II ->Z-HUB EINGEFAHREN
      )     ;
      U(    ;
      O     "I_WW_X_inWartePos"; // X-ACHSE IST AUF WARTEPOSITION
      O     "M_WW_X_imArbeitsraum"; // X-ACHSE NICHT IM WZW
      )     ;
      U     "DB_WW".Schritt_T[2]; // SCHRITT2 MAGPOS, WZ-ZANGE AUF
      U     #Schritt_rueckwaerts; // SCHRITTKETTE RUECKWAERTS

      S     "DB_WW".Schritt_T[1]; // SCHRITT1 WARTEPOS, RICHTEN, WZ-ENTSPANNE
      R     "DB_WW".Schritt_T[0]; // SCHRITT0 GRUNDSTELLUNG
      R     "DB_WW".Schritt_T[2]; // SCHRITT2 MAGPOS, WZ-ZANGE AUF

NETWORK
TITLE =WW: SCHRITT_2
// VORW.AUFTRAG1,3: X-ACHSE MAGPOS ANFAHREN
// RUECK.AUFTRAG1 : X-ACHSE WARTEPOS ANFAHREN
// RUECK.AUFTRAG3 : WZ-ZANGE SCHLIESSEN, X-ACHSE WARTEPOS ANFAHREN
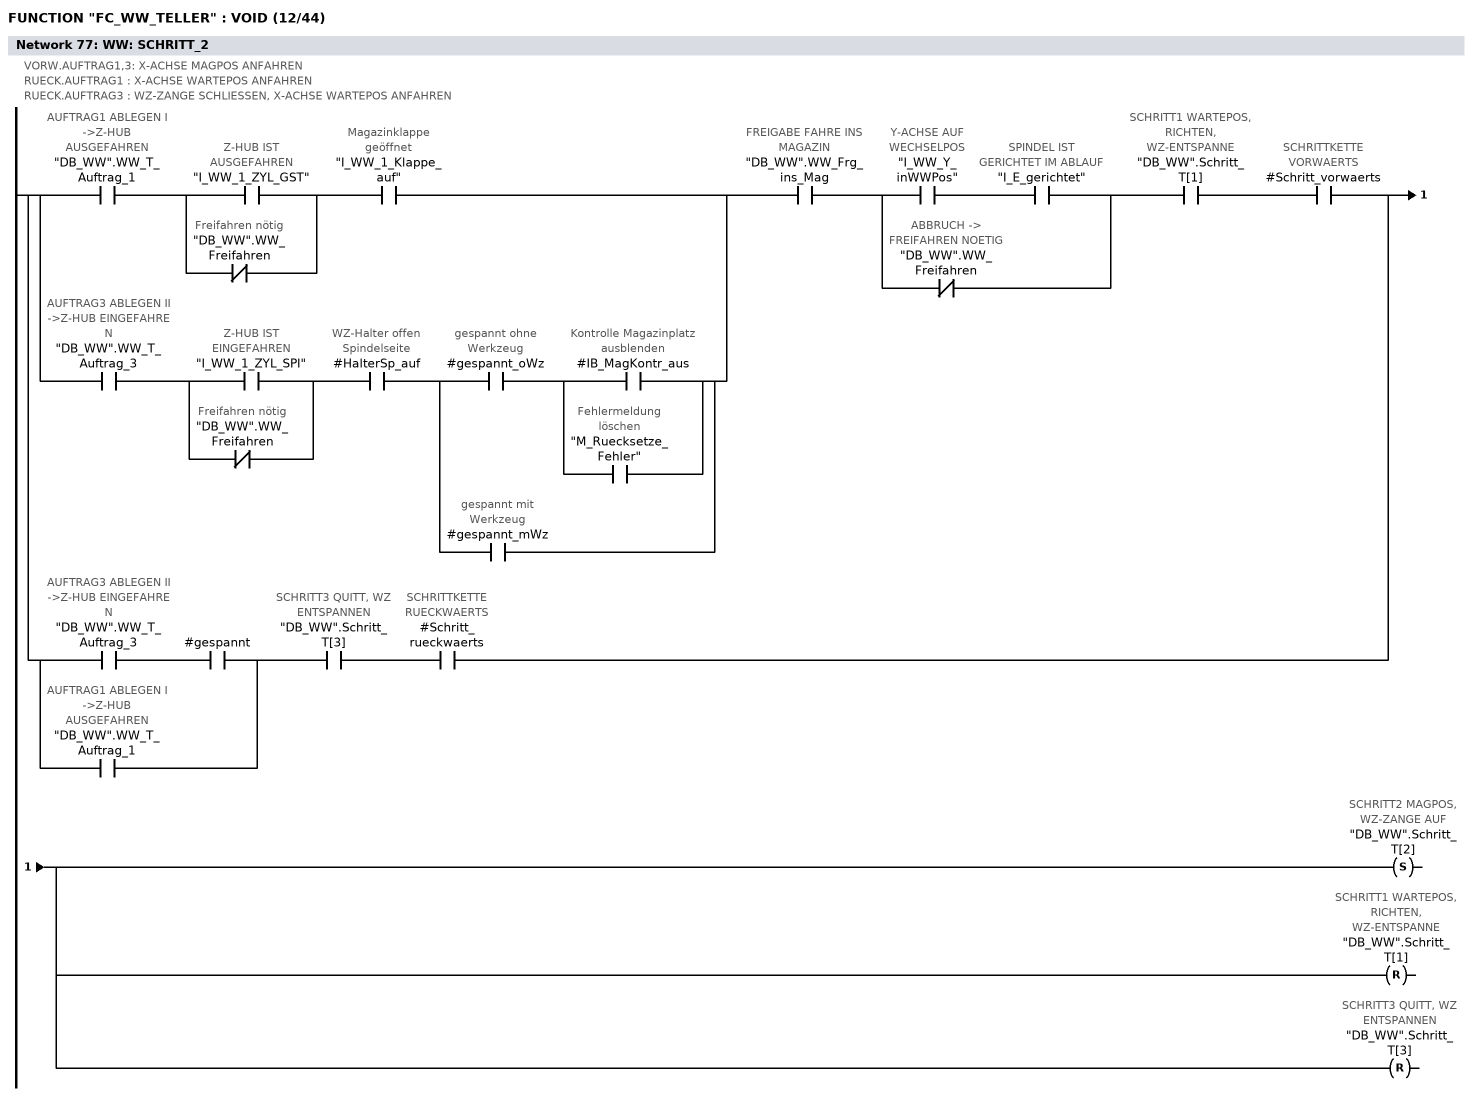
      U(    ;
      U     "DB_WW".WW_T_Auftrag_1; // AUFTRAG1 ABLEGEN I ->Z-HUB AUSGEFAHREN
      U(    ;
      O     "I_WW_1_ZYL_GST"; // Z-HUB IST AUSGEFAHREN
      ON    "DB_WW".WW_Freifahren; // Freifahren nötig
      )     ;
      U     "I_WW_1_Klappe_auf"; // Magazinklappe geöffnet
      O     ;
      U     "DB_WW".WW_T_Auftrag_3; // AUFTRAG3 ABLEGEN II ->Z-HUB EINGEFAHREN
      U(    ;
      O     "I_WW_1_ZYL_SPI"; // Z-HUB IST EINGEFAHREN
      ON    "DB_WW".WW_Freifahren; // Freifahren nötig
      )     ;
      U     #HalterSp_auf; // WZ-Halter offen Spindelseite
      U(    ;
      U     #gespannt_oWz; // gespannt ohne Werkzeug
      U(    ;
      O     #IB_MagKontr_aus; // Kontrolle Magazinplatz ausblenden
      O     "M_Ruecksetze_Fehler"; // Fehlermeldung löschen
      )     ;
      O     #gespannt_mWz; // gespannt mit Werkzeug
      )     ;
      )     ;
      U     "DB_WW".WW_Frg_ins_Mag; // FREIGABE FAHRE INS MAGAZIN
      U(    ;
      U     "I_WW_Y_inWWPos"; // Y-ACHSE AUF WECHSELPOS
      U     "I_E_gerichtet"; // SPINDEL IST GERICHTET IM ABLAUF
      ON    "DB_WW".WW_Freifahren; // ABBRUCH -> FREIFAHREN NOETIG
      )     ;
      U     "DB_WW".Schritt_T[1]; // SCHRITT1 WARTEPOS, RICHTEN, WZ-ENTSPANNE
      U     #Schritt_vorwaerts; // SCHRITTKETTE VORWAERTS

      O     ;
      U(    ;
      U     "DB_WW".WW_T_Auftrag_3; // AUFTRAG3 ABLEGEN II ->Z-HUB EINGEFAHREN
      U     #gespannt;
//      U     #gespannt_mWz               // gespannt mit Werkzeug
      O     "DB_WW".WW_T_Auftrag_1; // AUFTRAG1 ABLEGEN I ->Z-HUB AUSGEFAHREN
      )     ;
      U     "DB_WW".Schritt_T[3]; // SCHRITT3 QUITT, WZ ENTSPANNEN
      U     #Schritt_rueckwaerts; // SCHRITTKETTE RUECKWAERTS

      S     "DB_WW".Schritt_T[2]; // SCHRITT2 MAGPOS, WZ-ZANGE AUF
      R     "DB_WW".Schritt_T[1]; // SCHRITT1 WARTEPOS, RICHTEN, WZ-ENTSPANNE
      R     "DB_WW".Schritt_T[3]; // SCHRITT3 QUITT, WZ ENTSPANNEN

NETWORK
TITLE =WW: SCHRITT_3
// VORW. AUFTRAG1 : QUITTIEREN
// VORW. AUFTRAG3 : WZ-SPANNER OEFFNEN, WZ-ZANGE SCHLIESSEN
// RUECK.AUFTRAG1 : QUITTIEREN
// RUECK.AUFTRAG3 : WZ-SPANNER SCHLIESSEN
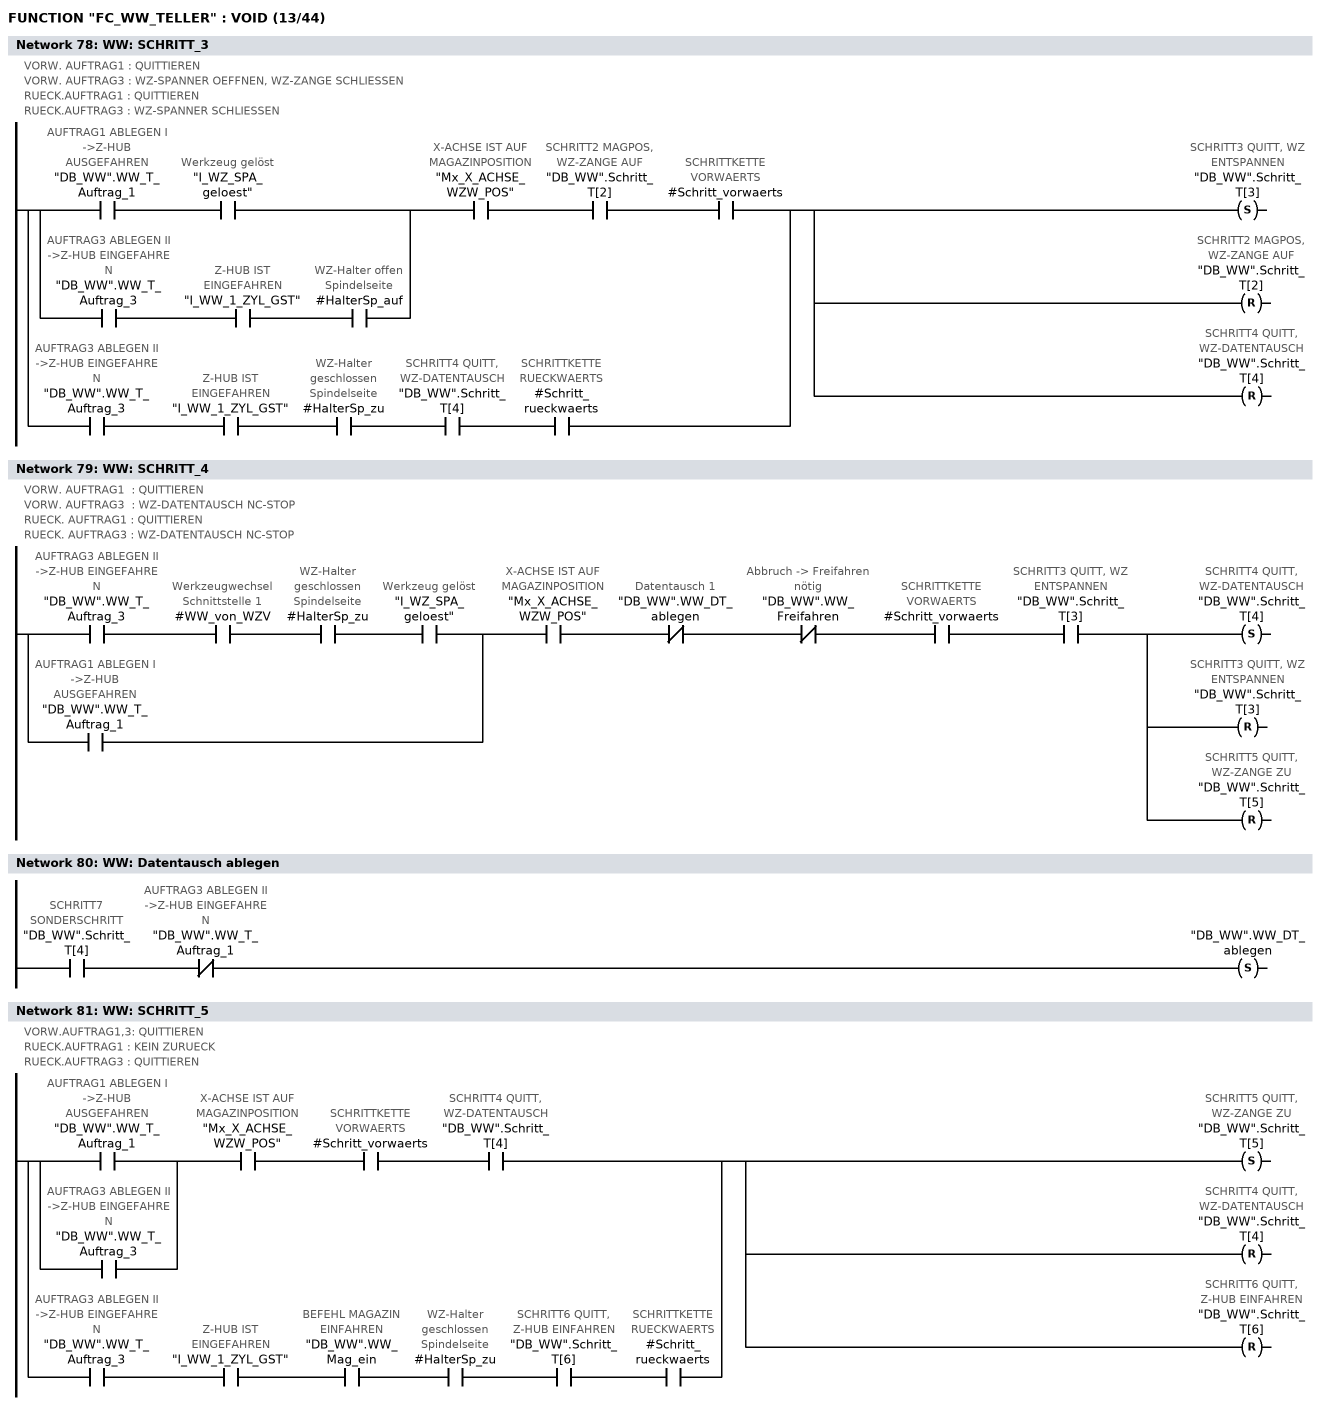
      U(    ;
      U     "DB_WW".WW_T_Auftrag_1; // AUFTRAG1 ABLEGEN I ->Z-HUB AUSGEFAHREN
      U     "I_WZ_SPA_geloest"; // Werkzeug gelöst
      O     ;
      U     "DB_WW".WW_T_Auftrag_3; // AUFTRAG3 ABLEGEN II ->Z-HUB EINGEFAHREN
      U     "I_WW_1_ZYL_GST"; // Z-HUB IST EINGEFAHREN
      U     #HalterSp_auf; // WZ-Halter offen Spindelseite
      )     ;
      U     "Mx_X_ACHSE_WZW_POS"; // X-ACHSE IST AUF MAGAZINPOSITION
      U     "DB_WW".Schritt_T[2]; // SCHRITT2 MAGPOS, WZ-ZANGE AUF
      U     #Schritt_vorwaerts; // SCHRITTKETTE VORWAERTS

      O     ;
      U     "DB_WW".WW_T_Auftrag_3; // AUFTRAG3 ABLEGEN II ->Z-HUB EINGEFAHREN
      U     "I_WW_1_ZYL_GST"; // Z-HUB IST EINGEFAHREN
      U     #HalterSp_zu; // WZ-Halter geschlossen Spindelseite
      U     "DB_WW".Schritt_T[4]; // SCHRITT4 QUITT, WZ-DATENTAUSCH
      U     #Schritt_rueckwaerts; // SCHRITTKETTE RUECKWAERTS

      S     "DB_WW".Schritt_T[3]; // SCHRITT3 QUITT, WZ ENTSPANNEN
      R     "DB_WW".Schritt_T[2]; // SCHRITT2 MAGPOS, WZ-ZANGE AUF
      R     "DB_WW".Schritt_T[4]; // SCHRITT4 QUITT, WZ-DATENTAUSCH

NETWORK
TITLE =WW: SCHRITT_4
// VORW. AUFTRAG1  : QUITTIEREN
// VORW. AUFTRAG3  : WZ-DATENTAUSCH NC-STOP
// RUECK. AUFTRAG1 : QUITTIEREN
// RUECK. AUFTRAG3 : WZ-DATENTAUSCH NC-STOP
      U(    ;
      U     "DB_WW".WW_T_Auftrag_3; // AUFTRAG3 ABLEGEN II ->Z-HUB EINGEFAHREN
      U     #WW_von_WZV; // Werkzeugwechsel Schnittstelle 1
      U     #HalterSp_zu; // WZ-Halter geschlossen Spindelseite
      U     "I_WZ_SPA_geloest"; // Werkzeug gelöst
      O     "DB_WW".WW_T_Auftrag_1; // AUFTRAG1 ABLEGEN I ->Z-HUB AUSGEFAHREN
      )     ;
      U     "Mx_X_ACHSE_WZW_POS"; // X-ACHSE IST AUF MAGAZINPOSITION
      UN    "DB_WW".WW_DT_ablegen; // Datentausch 1
      UN    "DB_WW".WW_Freifahren; // Abbruch -> Freifahren nötig
      U     #Schritt_vorwaerts; // SCHRITTKETTE VORWAERTS
      U     "DB_WW".Schritt_T[3]; // SCHRITT3 QUITT, WZ ENTSPANNEN
      S     "DB_WW".Schritt_T[4]; // SCHRITT4 QUITT, WZ-DATENTAUSCH
      R     "DB_WW".Schritt_T[3]; // SCHRITT3 QUITT, WZ ENTSPANNEN
      R     "DB_WW".Schritt_T[5]; // SCHRITT5 QUITT, WZ-ZANGE ZU

NETWORK
TITLE =WW: Datentausch ablegen

      U     "DB_WW".Schritt_T[4]; // SCHRITT7 SONDERSCHRITT
      UN    "DB_WW".WW_T_Auftrag_1; // AUFTRAG3 ABLEGEN II ->Z-HUB EINGEFAHREN
      S     "DB_WW".WW_DT_ablegen;


NETWORK
TITLE =WW: SCHRITT_5
// VORW.AUFTRAG1,3: QUITTIEREN
// RUECK.AUFTRAG1 : KEIN ZURUECK
// RUECK.AUFTRAG3 : QUITTIEREN
      U(    ;
      O     "DB_WW".WW_T_Auftrag_1; // AUFTRAG1 ABLEGEN I ->Z-HUB AUSGEFAHREN
      O     "DB_WW".WW_T_Auftrag_3; // AUFTRAG3 ABLEGEN II ->Z-HUB EINGEFAHREN
      )     ;
      U     "Mx_X_ACHSE_WZW_POS"; // X-ACHSE IST AUF MAGAZINPOSITION
      U     #Schritt_vorwaerts; // SCHRITTKETTE VORWAERTS
      U     "DB_WW".Schritt_T[4]; // SCHRITT4 QUITT, WZ-DATENTAUSCH
      O     ;
      U     "DB_WW".WW_T_Auftrag_3; // AUFTRAG3 ABLEGEN II ->Z-HUB EINGEFAHREN
      U     "I_WW_1_ZYL_GST"; // Z-HUB IST EINGEFAHREN
      U     "DB_WW".WW_Mag_ein; // BEFEHL MAGAZIN EINFAHREN
      U     #HalterSp_zu; // WZ-Halter geschlossen Spindelseite
      U     "DB_WW".Schritt_T[6]; // SCHRITT6 QUITT, Z-HUB EINFAHREN
      U     #Schritt_rueckwaerts; // SCHRITTKETTE RUECKWAERTS
      S     "DB_WW".Schritt_T[5]; // SCHRITT5 QUITT, WZ-ZANGE ZU
      R     "DB_WW".Schritt_T[4]; // SCHRITT4 QUITT, WZ-DATENTAUSCH
      R     "DB_WW".Schritt_T[6]; // SCHRITT6 QUITT, Z-HUB EINFAHREN

NETWORK
TITLE =WW: SCHRITT_6
// VORW.AUFTRAG1   : QUITTIEREN
// VORW.AUFTRAG3   : Z-HUB AUSFAHREN
// RUECK.AUFTRAG1,3: KEIN ZURUECK
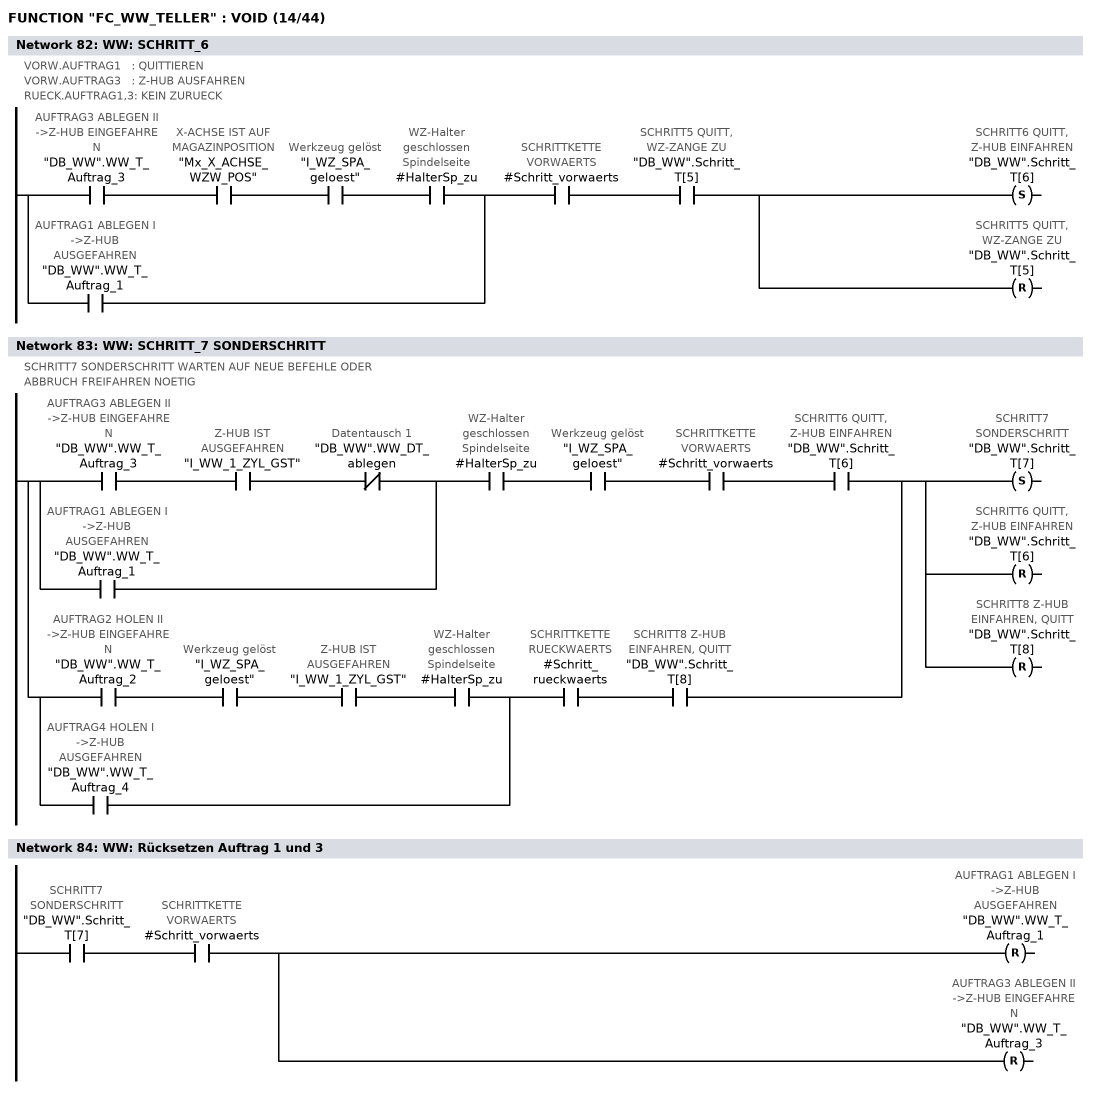
      U(    ;
      U     "DB_WW".WW_T_Auftrag_3; // AUFTRAG3 ABLEGEN II ->Z-HUB EINGEFAHREN
      U     "Mx_X_ACHSE_WZW_POS"; // X-ACHSE IST AUF MAGAZINPOSITION
      U     "I_WZ_SPA_geloest"; // Werkzeug gelöst
      U     #HalterSp_zu; // WZ-Halter geschlossen Spindelseite
      O     "DB_WW".WW_T_Auftrag_1; // AUFTRAG1 ABLEGEN I ->Z-HUB AUSGEFAHREN
      )     ;
      U     #Schritt_vorwaerts; // SCHRITTKETTE VORWAERTS
      U     "DB_WW".Schritt_T[5]; // SCHRITT5 QUITT, WZ-ZANGE ZU
      S     "DB_WW".Schritt_T[6]; // SCHRITT6 QUITT, Z-HUB EINFAHREN
      R     "DB_WW".Schritt_T[5]; // SCHRITT5 QUITT, WZ-ZANGE ZU

NETWORK
TITLE =WW: SCHRITT_7 SONDERSCHRITT
// SCHRITT7 SONDERSCHRITT WARTEN AUF NEUE BEFEHLE ODER
//                        ABBRUCH FREIFAHREN NOETIG
      U(    ;
      U     "DB_WW".WW_T_Auftrag_3; // AUFTRAG3 ABLEGEN II ->Z-HUB EINGEFAHREN
      U     "I_WW_1_ZYL_GST"; // Z-HUB IST AUSGEFAHREN
      UN    "DB_WW".WW_DT_ablegen; // Datentausch 1
      O     "DB_WW".WW_T_Auftrag_1; // AUFTRAG1 ABLEGEN I ->Z-HUB AUSGEFAHREN
      )     ;
      U     #HalterSp_zu; // WZ-Halter geschlossen Spindelseite
      U     "I_WZ_SPA_geloest"; // Werkzeug gelöst
      U     #Schritt_vorwaerts; // SCHRITTKETTE VORWAERTS
      U     "DB_WW".Schritt_T[6]; // SCHRITT6 QUITT, Z-HUB EINFAHREN
      O     ;
      U(    ;
      U     "DB_WW".WW_T_Auftrag_2; // AUFTRAG2 HOLEN II ->Z-HUB EINGEFAHREN
      U     "I_WZ_SPA_geloest"; // Werkzeug gelöst
      U     "I_WW_1_ZYL_GST"; // Z-HUB IST AUSGEFAHREN
      U     #HalterSp_zu; // WZ-Halter geschlossen Spindelseite
      O     "DB_WW".WW_T_Auftrag_4; // AUFTRAG4 HOLEN I ->Z-HUB AUSGEFAHREN
      )     ;
      U     #Schritt_rueckwaerts; // SCHRITTKETTE RUECKWAERTS
      U     "DB_WW".Schritt_T[8]; // SCHRITT8 Z-HUB EINFAHREN, QUITT
      S     "DB_WW".Schritt_T[7]; // SCHRITT7 SONDERSCHRITT
      R     "DB_WW".Schritt_T[6]; // SCHRITT6 QUITT, Z-HUB EINFAHREN
      R     "DB_WW".Schritt_T[8]; // SCHRITT8 Z-HUB EINFAHREN, QUITT

NETWORK
TITLE =WW: Rücksetzen Auftrag 1 und 3

      U     "DB_WW".Schritt_T[7]; // SCHRITT7 SONDERSCHRITT
      U     #Schritt_vorwaerts; // SCHRITTKETTE VORWAERTS
      R     "DB_WW".WW_T_Auftrag_1; // AUFTRAG1 ABLEGEN I ->Z-HUB AUSGEFAHREN
      R     "DB_WW".WW_T_Auftrag_3; // AUFTRAG3 ABLEGEN II ->Z-HUB EINGEFAHREN

NETWORK
TITLE =WW: SCHRITT_8
// VORW.AUFTRAG2  : Z-HUB EINFAHREN
// VORW.AUFTRAG4  : QUITTIEREN
// RUECK.AUFTRAG2 : Z-HUB AUSFAHREN
// RUECK.AUFTRAG4 : QUITTIEREN
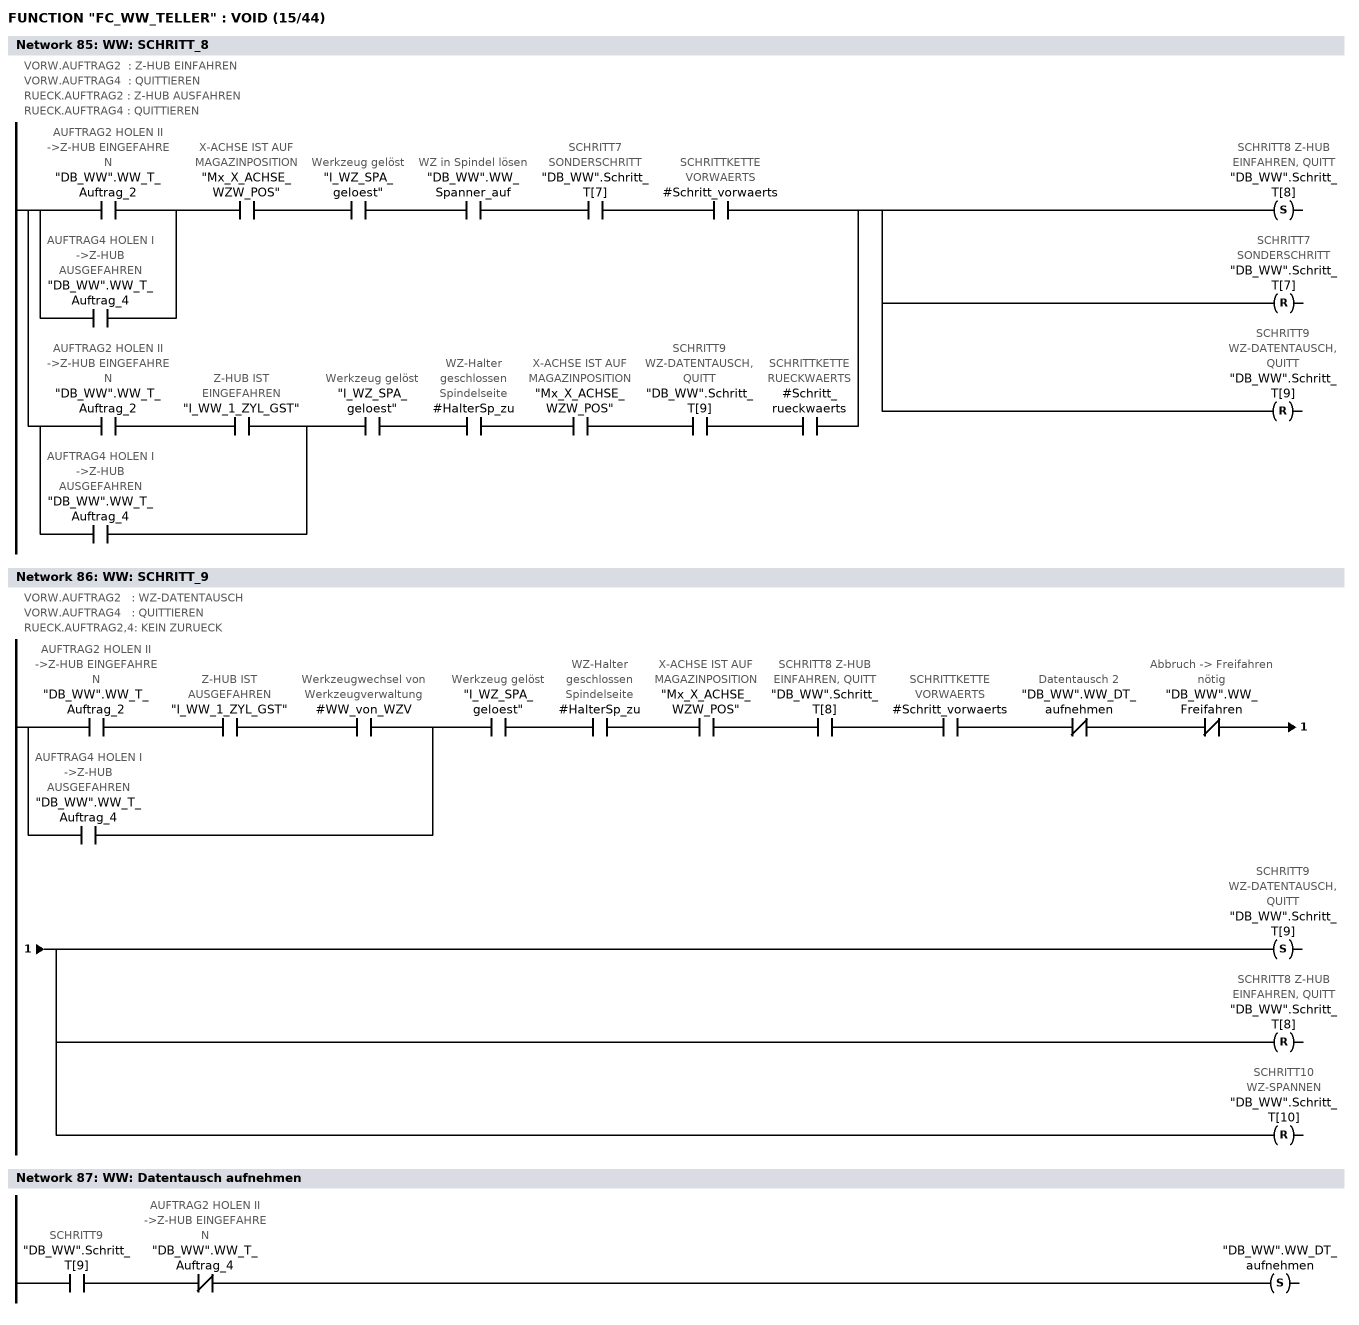
      U(    ;
      O     "DB_WW".WW_T_Auftrag_2; // AUFTRAG2 HOLEN II ->Z-HUB EINGEFAHREN
      O     "DB_WW".WW_T_Auftrag_4; // AUFTRAG4 HOLEN I ->Z-HUB AUSGEFAHREN
      )     ;
      U     "Mx_X_ACHSE_WZW_POS"; // X-ACHSE IST AUF MAGAZINPOSITION
      U     "I_WZ_SPA_geloest"; // Werkzeug gelöst
      U     "DB_WW".WW_Spanner_auf; // WZ in Spindel lösen
      U     "DB_WW".Schritt_T[7]; // SCHRITT7 SONDERSCHRITT
      U     #Schritt_vorwaerts; // SCHRITTKETTE VORWAERTS
      O     ;
      U(    ;
      U     "DB_WW".WW_T_Auftrag_2; // AUFTRAG2 HOLEN II ->Z-HUB EINGEFAHREN
      U     "I_WW_1_ZYL_GST"; // Z-HUB IST EINGEFAHREN
      O     "DB_WW".WW_T_Auftrag_4; // AUFTRAG4 HOLEN I ->Z-HUB AUSGEFAHREN
      )     ;
      U     "I_WZ_SPA_geloest"; // Werkzeug gelöst
      U     #HalterSp_zu; // WZ-Halter geschlossen Spindelseite
      U     "Mx_X_ACHSE_WZW_POS"; // X-ACHSE IST AUF MAGAZINPOSITION
      U     "DB_WW".Schritt_T[9]; // SCHRITT9 WZ-DATENTAUSCH, QUITT
      U     #Schritt_rueckwaerts; // SCHRITTKETTE RUECKWAERTS
      S     "DB_WW".Schritt_T[8]; // SCHRITT8 Z-HUB EINFAHREN, QUITT
      R     "DB_WW".Schritt_T[7]; // SCHRITT7 SONDERSCHRITT
      R     "DB_WW".Schritt_T[9]; // SCHRITT9 WZ-DATENTAUSCH, QUITT

NETWORK
TITLE =WW: SCHRITT_9
// VORW.AUFTRAG2   : WZ-DATENTAUSCH
// VORW.AUFTRAG4   : QUITTIEREN
// RUECK.AUFTRAG2,4: KEIN ZURUECK
      U(    ;
      U     "DB_WW".WW_T_Auftrag_2; // AUFTRAG2 HOLEN II ->Z-HUB EINGEFAHREN
      U     "I_WW_1_ZYL_GST"; // Z-HUB IST AUSGEFAHREN
      U     #WW_von_WZV; // Werkzeugwechsel von Werkzeugverwaltung
      O     "DB_WW".WW_T_Auftrag_4; // AUFTRAG4 HOLEN I ->Z-HUB AUSGEFAHREN
      )     ;
      U     "I_WZ_SPA_geloest"; // Werkzeug gelöst
      U     #HalterSp_zu; // WZ-Halter geschlossen Spindelseite
      U     "Mx_X_ACHSE_WZW_POS"; // X-ACHSE IST AUF MAGAZINPOSITION
      U     "DB_WW".Schritt_T[8]; // SCHRITT8 Z-HUB EINFAHREN, QUITT
      U     #Schritt_vorwaerts; // SCHRITTKETTE VORWAERTS
      UN    "DB_WW".WW_DT_aufnehmen; // Datentausch 2
      UN    "DB_WW".WW_Freifahren; // Abbruch -> Freifahren nötig
      S     "DB_WW".Schritt_T[9]; // SCHRITT9 WZ-DATENTAUSCH, QUITT
      R     "DB_WW".Schritt_T[8]; // SCHRITT8 Z-HUB EINFAHREN, QUITT
      R     "DB_WW".Schritt_T[10]; // SCHRITT10 WZ-SPANNEN

NETWORK
TITLE =WW: Datentausch aufnehmen

      U     "DB_WW".Schritt_T[9]; // SCHRITT9
      UN    "DB_WW".WW_T_Auftrag_4; // AUFTRAG2 HOLEN II ->Z-HUB EINGEFAHREN
      S     "DB_WW".WW_DT_aufnehmen;

NETWORK
TITLE =WW: SCHRITT_10
// VORW.AUFTRAG2    : WZ-SPANNEN, WZ-ZANGE OEFFNEN
// VORW.Auftrag4    : WZ-SPANNEN
// RUECK.AUFTRAG2,4 : KEIN ZURUECK
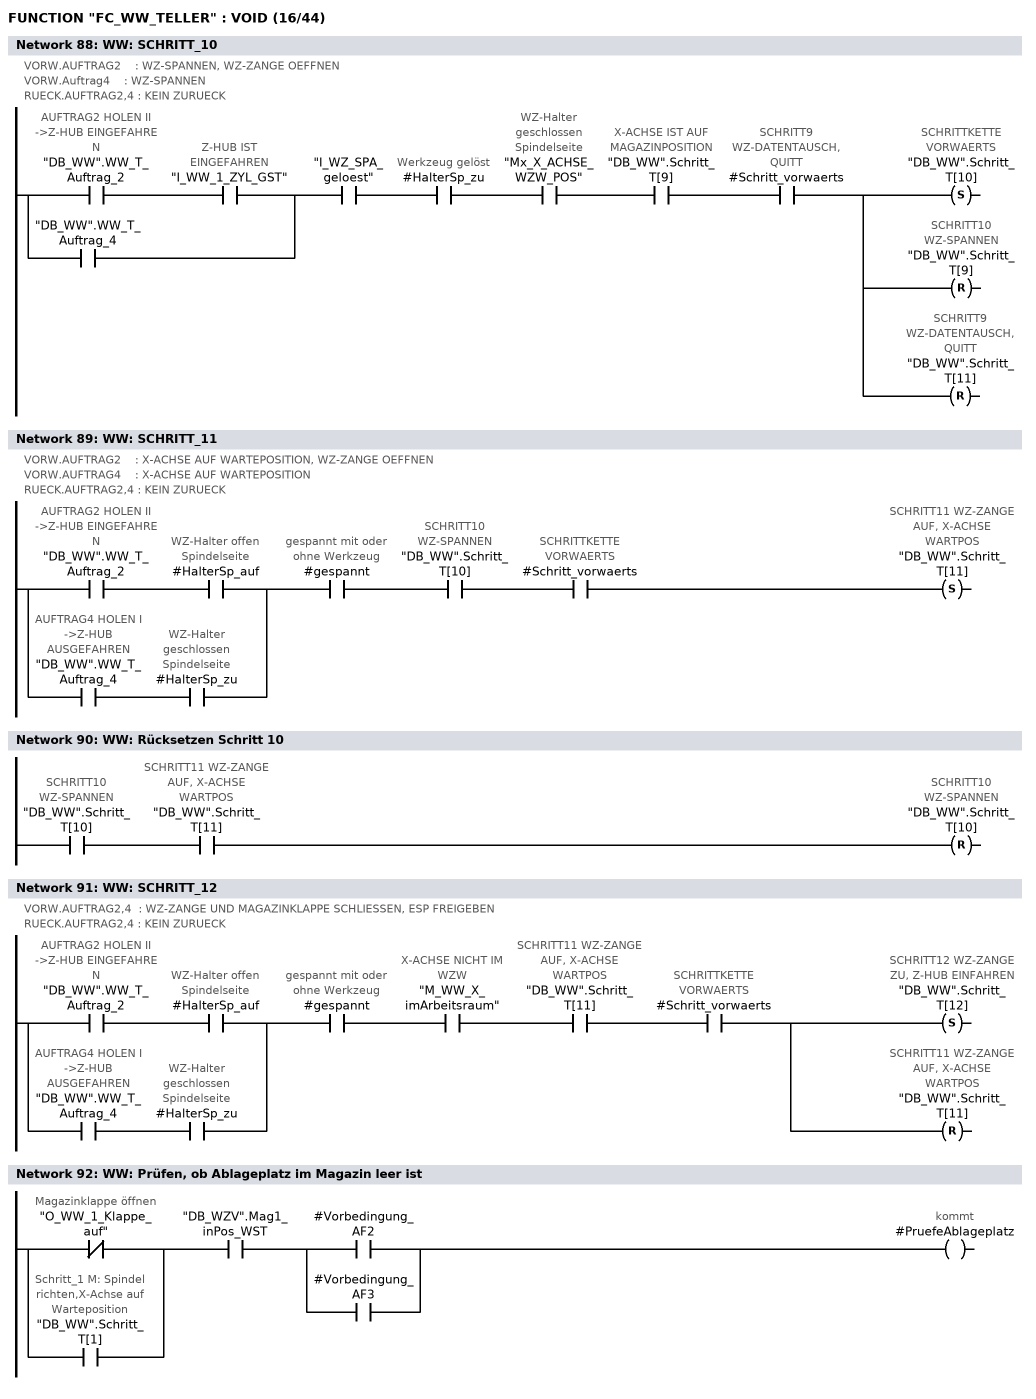
      U(    ;
      U     "DB_WW".WW_T_Auftrag_2; // AUFTRAG2 HOLEN II ->Z-HUB EINGEFAHREN
      U     "I_WW_1_ZYL_GST"; // Z-HUB IST EINGEFAHREN
      O     "DB_WW".WW_T_Auftrag_4;
      )     ; // AUFTRAG4 HOLEN I ->Z-HUB AUSGEFAHREN
      U     "I_WZ_SPA_geloest";
      U     #HalterSp_zu; // Werkzeug gelöst
      U     "Mx_X_ACHSE_WZW_POS"; // WZ-Halter geschlossen Spindelseite
      U     "DB_WW".Schritt_T[9]; // X-ACHSE IST AUF MAGAZINPOSITION
      U     #Schritt_vorwaerts; // SCHRITT9 WZ-DATENTAUSCH, QUITT
      S     "DB_WW".Schritt_T[10]; // SCHRITTKETTE VORWAERTS
      R     "DB_WW".Schritt_T[9]; // SCHRITT10 WZ-SPANNEN
      R     "DB_WW".Schritt_T[11]; // SCHRITT9 WZ-DATENTAUSCH, QUITT
NETWORK
TITLE =WW: SCHRITT_11
// VORW.AUFTRAG2    : X-ACHSE AUF WARTEPOSITION, WZ-ZANGE OEFFNEN
// VORW.AUFTRAG4    : X-ACHSE AUF WARTEPOSITION
// RUECK.AUFTRAG2,4 : KEIN ZURUECK
      U(    ;
      U     "DB_WW".WW_T_Auftrag_2; // AUFTRAG2 HOLEN II ->Z-HUB EINGEFAHREN
      U     #HalterSp_auf; // WZ-Halter offen Spindelseite
      O     ;
      U     "DB_WW".WW_T_Auftrag_4; // AUFTRAG4 HOLEN I ->Z-HUB AUSGEFAHREN
      U     #HalterSp_zu; // WZ-Halter geschlossen Spindelseite
      )     ;
      U     #gespannt; // gespannt mit oder ohne Werkzeug
      U     "DB_WW".Schritt_T[10]; // SCHRITT10 WZ-SPANNEN
      U     #Schritt_vorwaerts; // SCHRITTKETTE VORWAERTS
      S     "DB_WW".Schritt_T[11]; // SCHRITT11 WZ-ZANGE AUF, X-ACHSE WARTPOS

NETWORK
TITLE =WW: Rücksetzen Schritt 10

      U     "DB_WW".Schritt_T[10]; // SCHRITT10 WZ-SPANNEN
      U     "DB_WW".Schritt_T[11]; // SCHRITT11 WZ-ZANGE AUF, X-ACHSE WARTPOS
      R     "DB_WW".Schritt_T[10]; // SCHRITT10 WZ-SPANNEN

NETWORK
TITLE =WW: SCHRITT_12
// VORW.AUFTRAG2,4  : WZ-ZANGE UND MAGAZINKLAPPE SCHLIESSEN, ESP FREIGEBEN
// RUECK.AUFTRAG2,4 : KEIN ZURUECK
      U(    ;
      U     "DB_WW".WW_T_Auftrag_2; // AUFTRAG2 HOLEN II ->Z-HUB EINGEFAHREN
      U     #HalterSp_auf; // WZ-Halter offen Spindelseite
      O     ;
      U     "DB_WW".WW_T_Auftrag_4; // AUFTRAG4 HOLEN I ->Z-HUB AUSGEFAHREN
      U     #HalterSp_zu; // WZ-Halter geschlossen Spindelseite
      )     ;
      U     #gespannt; // gespannt mit oder ohne Werkzeug
      U     "M_WW_X_imArbeitsraum"; // X-ACHSE NICHT IM WZW
      U     "DB_WW".Schritt_T[11]; // SCHRITT11 WZ-ZANGE AUF, X-ACHSE WARTPOS
      U     #Schritt_vorwaerts; // SCHRITTKETTE VORWAERTS
      S     "DB_WW".Schritt_T[12]; // SCHRITT12 WZ-ZANGE ZU, Z-HUB EINFAHREN
      R     "DB_WW".Schritt_T[11]; // SCHRITT11 WZ-ZANGE AUF, X-ACHSE WARTPOS

NETWORK
TITLE =WW: Prüfen, ob Ablageplatz im Magazin leer ist

      U(    ;
      ON    "O_WW_1_Klappe_auf"; // Magazinklappe öffnen
      O     "DB_WW".Schritt_T[1]; // Schritt_1 M: Spindel richten,X-Achse auf Warteposition
      )     ;
      U     "DB_WZV".Mag1_inPos_WST;
      U(    ;
      O     #Vorbedingung_AF2;
      O     #Vorbedingung_AF3;
      )     ;
      =     #PruefeAblageplatz; // kommt

NETWORK
TITLE =WW: Prüfen, ob Abholplatz im Magazin belegt ist
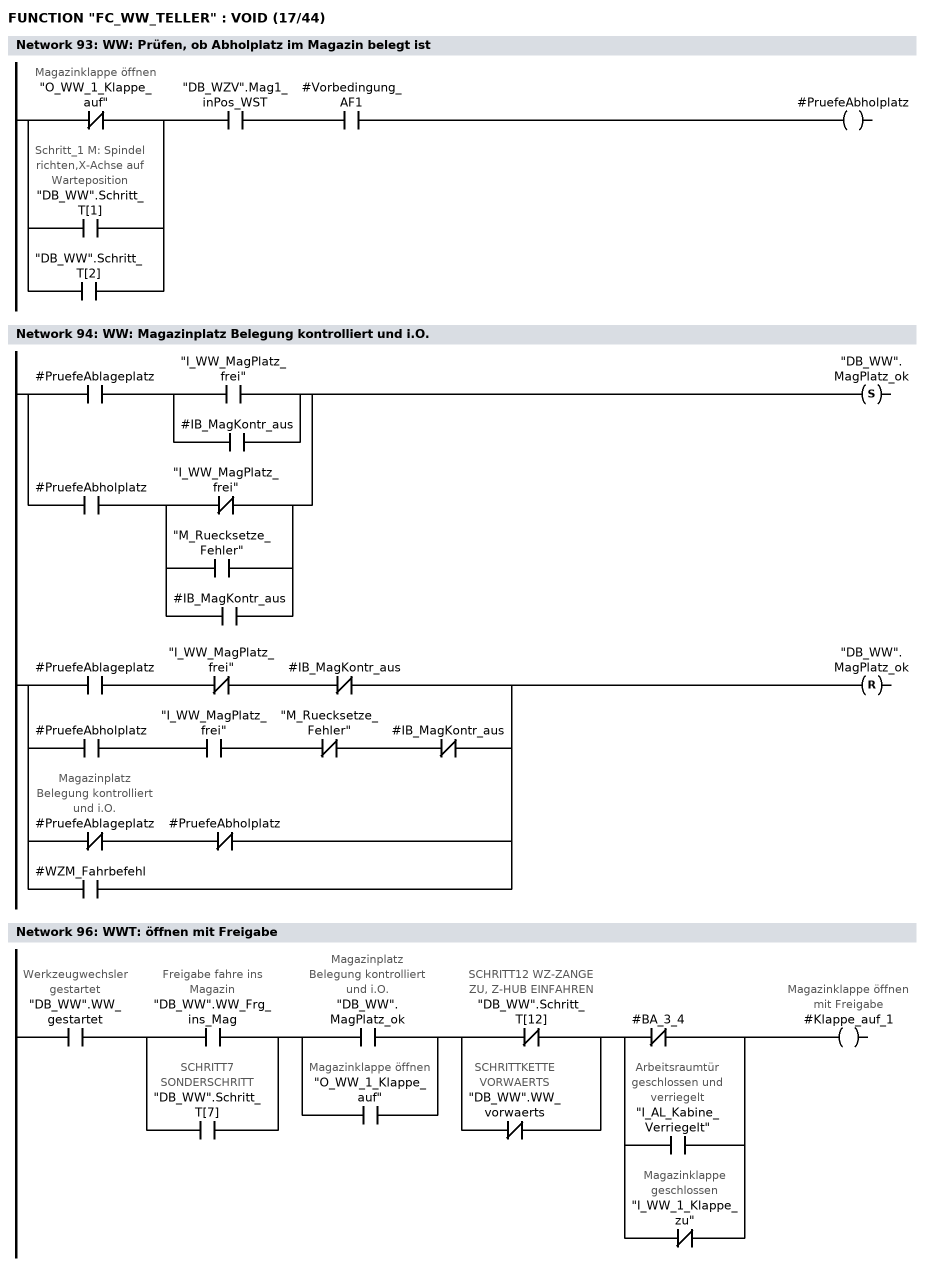

      U(    ;
      ON    "O_WW_1_Klappe_auf"; // Magazinklappe öffnen
      O     "DB_WW".Schritt_T[1]; // Schritt_1 M: Spindel richten,X-Achse auf Warteposition
      O     "DB_WW".Schritt_T[2];
      )     ;
      U     "DB_WZV".Mag1_inPos_WST;
      U     #Vorbedingung_AF1;
      =     #PruefeAbholplatz;

NETWORK
TITLE =WW: Magazinplatz Belegung kontrolliert und i.O.

      U(    ;
      U     #PruefeAblageplatz;
      U(    ;
      O     "I_WW_MagPlatz_frei";
      O     #IB_MagKontr_aus;
      )     ;
      O     ;
      U     #PruefeAbholplatz;
      U(    ;
      ON    "I_WW_MagPlatz_frei";
      O     "M_Ruecksetze_Fehler";
      O     #IB_MagKontr_aus;
      )     ;
      )     ;
      S     "DB_WW".MagPlatz_ok;

      U(    ;
      U     #PruefeAblageplatz;
      UN    "I_WW_MagPlatz_frei";
      UN    #IB_MagKontr_aus;
      O     ;
      U     #PruefeAbholplatz;
      U     "I_WW_MagPlatz_frei";
      UN    "M_Ruecksetze_Fehler";
      UN    #IB_MagKontr_aus;
      O     ;
      UN    #PruefeAblageplatz; // Magazinplatz Belegung kontrolliert und i.O.
      UN    #PruefeAbholplatz;

      O     #WZM_Fahrbefehl;
      )     ;
      R     "DB_WW".MagPlatz_ok;
      NOP   0;
NETWORK
TITLE ============ Magazinklappe (Werkzeugwechslertür) =============



NETWORK
TITLE =WWT: öffnen mit Freigabe

      U     "DB_WW".WW_gestartet; // Werkzeugwechsler gestartet
      U(    ;
      O     "DB_WW".WW_Frg_ins_Mag; // Freigabe fahre ins Magazin
      O     "DB_WW".Schritt_T[7]; // SCHRITT7 SONDERSCHRITT
      )     ;

// Die Magazinklappe darf nur geöffnet werden, wenn der Magazinplatz kontrolliert wurde

      U(    ;
      O     "DB_WW".MagPlatz_ok; // Magazinplatz Belegung kontrolliert und i.O.
      O     "O_WW_1_Klappe_auf"; // Magazinklappe öffnen
      )     ;

// Klappe schliessen im Schritt 12 bei vorwärts
      U(    ;
      ON    "DB_WW".Schritt_T[12]; // SCHRITT12 WZ-ZANGE ZU, Z-HUB EINFAHREN
      ON    "DB_WW".WW_vorwaerts; // SCHRITTKETTE VORWAERTS
      )     ;

// Kein Öffnen der Klappe in BA3,4 solange die Magazinklappe geschlossen ist
      U(    ;
      ON    #BA_3_4;
      O     "I_AL_Kabine_Verriegelt"; // Arbeitsraumtür geschlossen und verriegelt
      ON    "I_WW_1_Klappe_zu"; // Magazinklappe geschlossen
      )     ;

      =     #Klappe_auf_1; // Magazinklappe öffnen mit Freigabe

NETWORK
TITLE =WWT: öffnen ohne Freigabe
